ABB RobotStudio station: OpenRobotica_versão16_03_V2.rspag

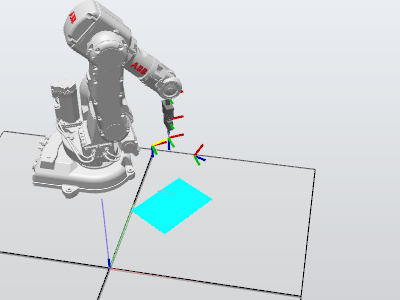
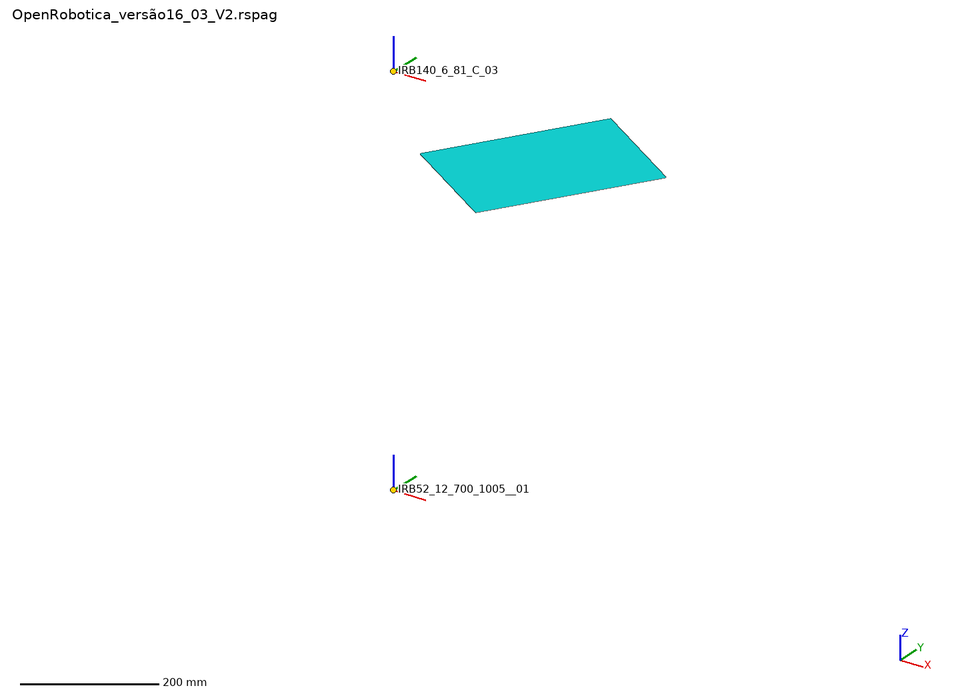
[picture v1: parts stored in the station drawn from their meshes, with robot base, taught points and paths (robot models come from the ABB library and are not in the file)]
--- station ---
Station V1 (saved by RobotStudio 23.2.10395.0)
Controller Robot_ISEP_IRB140, task T_ROB1: task frame (RAPID world) sits at (0, 0, 670) mm in the station
Controller Robot_ISEP_IRB140
  mechanical unit ROB_1: IRB140_6_81_C_03, 6 joints, base frame (0, 0, 0) mm
Controller Robo_open_v2
  mechanical unit ROB_1: IRB52_12_700_1005__01, 6 joints, base frame (0, 0, 0) mm, rotated rx 0 ry 0 rz 90 deg
Layout (positions relative to the parent item):
  - IRB140_6_81_C_03 [mechanism, from %ABB.RobotStudio.Models.IRB140%\IRB140_6_81_C_G_03.rslib] at (0, 0, 670) mm; joint values [0.4681, 0.0159, 0.7824, 0.0025, 0.7739, 3.0595] (rad or m)
  - rob-table [part, from Libraries\rob-table.rslib]
  - pen [mechanism, from Libraries\pen.rslib] at (0, 0, 0) mm
  - paper [part, from Libraries\paper.rslib]
  - IRB52_12_700_1005__01 [mechanism, from %ABB.RobotStudio.Models.IRB52%\IRB52_12_700_1005_G_01.rslib] at (0, 0, 0) mm, rotated rx 0 ry 0 rz 90 deg; joint values [0, 0, 0, 0, 0, 0] (rad or m)
  - A3_Vertical [part] at (450, 125, 790) mm, rotated rx 0 ry 0 rz -90 deg, size 297 x 420 x 0.5 mm
  - A3_Horizontal [part] at (747, 125, 790) mm, rotated rx 0 ry 0 rz 180 deg, size 297 x 420 x 0.5 mm
  - A4_Vertical [part] at (450, 125, 790) mm, rotated rx 0 ry 0 rz -90 deg, size 210 x 297 x 0.5 mm
  - A4_Horizontal [part] at (383.64, -3.77, 703.99) mm, rotated rx -179.83 ry -0.08 rz -32.58 deg, size 210 x 297 x 0.5 mm
  - A5_Vertical [part] at (450, 125, 790) mm, rotated rx 0 ry 0 rz -90 deg, size 148 x 210 x 0.5 mm
  - A5_Horizontal [part] at (450, -85, 790) mm, size 148 x 210 x 0.5 mm
  - MyNewTool [mechanism, from Libraries\Tool_IRB120.rslib] at (304.13, 153.88, 1044.81) mm, rotated rx -179.89 ry 0.07 rz 31.42 deg
Attachment: MyNewTool is attached to IRB140_6_81_C_03 / Link6
Targets, tools, work objects and paths stored in the station and not in the controller backup, written as RAPID:
! task T_ROB1
MODULE Module1
  CONST robtarget Target_Start:=[[0,0,0],[1,0,0,0],[0,0,0,0],[9E+09,9E+09,9E+09,9E+09,9E+09,9E+09]];
ENDMODULE

! task T_ROB1
MODULE DryLetter
  VAR robtarget sup_centro:=[[0,0,0],[1,0,0,0],[0,0,0,0],[9E+09,9E+09,9E+09,9E+09,9E+09,9E+09]];
  VAR robtarget meio_centro:=[[0,0,0],[1,0,0,0],[0,0,0,0],[9E+09,9E+09,9E+09,9E+09,9E+09,9E+09]];
  VAR robtarget inf_centro:=[[0,0,0],[1,0,0,0],[0,0,0,0],[9E+09,9E+09,9E+09,9E+09,9E+09,9E+09]];
  VAR robtarget up_meio_esq:=[[0,0,0],[1,0,0,0],[0,0,0,0],[9E+09,9E+09,9E+09,9E+09,9E+09,9E+09]];
  VAR robtarget sup_dir_meio:=[[0,0,0],[1,0,0,0],[0,0,0,0],[9E+09,9E+09,9E+09,9E+09,9E+09,9E+09]];
  VAR robtarget inf_dir_meio:=[[0,0,0],[1,0,0,0],[0,0,0,0],[9E+09,9E+09,9E+09,9E+09,9E+09,9E+09]];
ENDMODULE

! task T_ROB1
MODULE Math
  PROC impressmenu()
    write_string;
    calculo_size;
    settingsTextMenu;
    settingsPageMenu;
    write_string;
    impress_mecanism;
  ENDPROC
ENDMODULE

! task T_ROB1
MODULE Menu
  PROC start_default()
    WaitTime 3;
  ENDPROC
  PROC principal_menu()
    menu_text;
    menu_paper;
  ENDPROC
  PROC automaticPrinting()
    calculateSizeLetterAutomated;
    calculateOrigin;
    impressMecanism;
  ENDPROC
ENDMODULE

! task T_ROB1
MODULE Fonts
  VAR robtarget target_aMidInf1Esq12:=[[0,0,0],[1,0,0,0],[0,0,0,0],[9E+09,9E+09,9E+09,9E+09,9E+09,9E+09]];
  VAR robtarget target_oMidInf1Esq12:=[[0,0,0],[1,0,0,0],[0,0,0,0],[9E+09,9E+09,9E+09,9E+09,9E+09,9E+09]];
  VAR robtarget target_oMidInf1Dir12:=[[0,0,0],[1,0,0,0],[0,0,0,0],[9E+09,9E+09,9E+09,9E+09,9E+09,9E+09]];
  VAR robtarget target_aMidInf1Dir12:=[[0,0,0],[1,0,0,0],[0,0,0,0],[9E+09,9E+09,9E+09,9E+09,9E+09,9E+09]];
ENDMODULE


--- Backups/Robot_ISEP_IRB140/RAPID/TASK1/PROGMOD/CalibData.mod ---
MODULE CalibData
    PERS tooldata tWeldGun:=[TRUE,[[125.800591275,0,391.268161315],[0.898794046,0,0.438371147,0]],[3,[0,0,100],[0,1,0,0],0,0,0]];
    TASK PERS wobjdata Workobject_Paper:= [FALSE,TRUE,"",[[207.804,202.871,30.7786],[0.000727564,-0.962645,-0.270763,0.000849984]],[[0,0,0],[1,0,0,0]]];

    PERS wobjdata WA5 := [FALSE,TRUE,"",[[207.804,202.871,30.7786],[0.000727564,-0.962645,-0.270763,0.000849984]],[[0,0,0],[1,0,0,0]]];
    PERS wobjdata WA4 := [FALSE,TRUE,"",[[317.336,-107.098,31.058],[0.00324698,-0.996995,0.0772792,0.00429133]],[[0,0,0],[1,0,0,0]]];

    !TASK PERS wobjdata wba4gr3:=[FALSE,TRUE,"",[[317.336,-107.098,31.058],[0.00324698,-0.996995,0.0772792,0.00429133]],[[0,0,0],[1,0,0,0]]];
	!TASK PERS wobjdata wba5gr3:= [FALSE,TRUE,"",[[207.804,202.871,30.7786],[0.000727564,-0.962645,-0.270763,0.000849984]],[[0,0,0],[1,0,0,0]]];


    CONST robtarget Origem:=[[0,0,0],[1,0,0,0],[0,0,0,0],[9E+09,9E+09,9E+09,9E+09,9E+09,9E+09]];
    CONST robtarget Default_position:=[[55,95,-102.5],[1,0,0,0],[0,0,0,0],[9E+09,9E+09,9E+09,9E+09,9E+09,9E+09]];
   ! PERS tooldata pen:=[TRUE,[[0,0,139],[1,0,0,0]],[0.5,[0,0,20],[1,0,0,0],0,0,0]];
    PERS tooldata tcptool:=[TRUE,[[-1.2328,3.617,241.774],[1,0,0,0]],[1,[0,0,125],[1,0,0,0],0,0,0]];
    PERS tooldata pen:=[TRUE,[[0,0,139],[1,0,0,0]],[0.5,[0,0,20],[1,0,0,0],0,0,0]];
    PERS tooldata pen_1:=[TRUE,[[0,0,139],[1,0,0,0]],[0.5,[0,0,20],[1,0,0,0],0,0,0]];
ENDMODULE

--- Backups/Robot_ISEP_IRB140/RAPID/TASK1/PROGMOD/DryLetter.mod ---
MODULE DryLetter
    VAR robtarget up_inf_esq1:=[[0,0,0],[1,0,0,0],[0,0,0,0],[9E+09,9E+09,9E+09,9E+09,9E+09,9E+09]];
    VAR robtarget inf_esq1:=[[0,0,0],[1,0,0,0],[0,0,0,0],[9E+09,9E+09,9E+09,9E+09,9E+09,9E+09]];
    VAR robtarget sup_esq:=[[0,0,0],[1,0,0,0],[0,0,0,0],[9E+09,9E+09,9E+09,9E+09,9E+09,9E+09]];
    VAR robtarget sup_dir:=[[0,0,0],[1,0,0,0],[0,0,0,0],[9E+09,9E+09,9E+09,9E+09,9E+09,9E+09]];
    VAR robtarget inf_dir2:=[[0,0,0],[1,0,0,0],[0,0,0,0],[9E+09,9E+09,9E+09,9E+09,9E+09,9E+09]];
    VAR robtarget up_inf_dir2:=[[0,0,0],[1,0,0,0],[0,0,0,0],[9E+09,9E+09,9E+09,9E+09,9E+09,9E+09]];
    VAR robtarget meio_dir:=[[0,0,0],[1,0,0,0],[0,0,0,0],[9E+09,9E+09,9E+09,9E+09,9E+09,9E+09]];
    VAR robtarget meio_esq:=[[0,0,0],[1,0,0,0],[0,0,0,0],[9E+09,9E+09,9E+09,9E+09,9E+09,9E+09]];
    VAR robtarget up_final:=[[0,0,0],[1,0,0,0],[0,0,0,0],[9E+09,9E+09,9E+09,9E+09,9E+09,9E+09]];
    PROC Path_b()

    ENDPROC
    PROC dry_letter_a()

    ENDPROC
    PROC Letra_A()
        MoveJ up_inf_esq1,v100,fine,tcptool\WObj:=Workobject_Paper;
        MoveL inf_esq1,v100,fine,tcptool\WObj:=Workobject_Paper;
        MoveL sup_esq,v100,z0,tcptool\WObj:=Workobject_Paper;
        MoveL sup_dir,v100,z0,tcptool\WObj:=Workobject_Paper;
        MoveL inf_dir2,v100,fine,tcptool\WObj:=Workobject_Paper;
        MoveL up_inf_dir2,v100,z0,tcptool\WObj:=Workobject_Paper;
        MoveL meio_dir,v100,z0,tcptool\WObj:=Workobject_Paper;
        MoveL meio_esq,v100,fine,tcptool\WObj:=Workobject_Paper;
        MoveL up_final,v100,z0,tcptool\WObj:=Workobject_Paper;
    ENDPROC
    PROC Letra_B()
        MoveJ target_oInf1Esq1,v100,fine,tcptool\WObj:=Workobject_Paper;
        MoveL target_oInf1Esq1,v100,fine,tcptool\WObj:=Workobject_Paper;
        MoveL target_oInf1Esq1,v100,fine,tcptool\WObj:=Workobject_Paper;
    ENDPROC
    PROC Letra_F()
        MoveJ up_inf_esq1,v100,fine,tcptool\WObj:=Workobject_Paper;
    ENDPROC
    PROC Space_letter()
        MoveJ target_oInf1Esq1,v100,fine,tcptool\WObj:=Workobject_Paper;
    ENDPROC
ENDMODULE

--- Backups/Robot_ISEP_IRB140/RAPID/TASK1/PROGMOD/Fonts.mod ---
MODULE Fonts

    ! Offset Z
    VAR num offsetZa := 10;
    VAR num offsetZo := 1;

    ! On the paper

    VAR robtarget target_oInf1Esq1;
    VAR robtarget target_oInf1Esq2;
    VAR robtarget target_oInf1Centro;
    VAR robtarget target_oInf1Dir1;
    VAR robtarget target_oInf1Dir2;

    VAR robtarget target_oInf2Esq1;
    VAR robtarget target_oInf2Esq2;
    VAR robtarget target_oInf2Centro;
    VAR robtarget target_oInf2Dir1;
    VAR robtarget target_oInf2Dir2;

    VAR robtarget target_oCentroEsq1;
    VAR robtarget target_oCentroEsq2;
    VAR robtarget target_oCentroCentro;
    VAR robtarget target_oCentroDir1;
    VAR robtarget target_oCentroDir2;

    VAR robtarget target_oSup1Esq1;
    VAR robtarget target_oSup1Esq2;
    VAR robtarget target_oSup1Centro;
    VAR robtarget target_oSup1Dir1;
    VAR robtarget target_oSup1Dir2;

    VAR robtarget target_oSup2Esq1;
    VAR robtarget target_oSup2Esq2;
    VAR robtarget target_oSup2Centro;
    VAR robtarget target_oSup2Dir1;
    VAR robtarget target_oSup2Dir2;

    ! Above the paper

    VAR robtarget target_aInf1Esq1;
    VAR robtarget target_aInf1Esq2;
    VAR robtarget target_aInf1Centro;
    VAR robtarget target_aInf1Dir1;
    VAR robtarget target_aInf1Dir2;

    VAR robtarget target_aInf2Esq1;
    VAR robtarget target_aInf2Esq2;
    VAR robtarget target_aInf2Centro;
    VAR robtarget target_aInf2Dir1;
    VAR robtarget target_aInf2Dir2;

    VAR robtarget target_aCentroEsq1;
    VAR robtarget target_aCentroEsq2;
    VAR robtarget target_aCentroCentro;
    VAR robtarget target_aCentroDir1;
    VAR robtarget target_aCentroDir2;

    VAR robtarget target_aSup1Esq1;
    VAR robtarget target_aSup1Esq2;
    VAR robtarget target_aSup1Centro;
    VAR robtarget target_aSup1Dir1;
    VAR robtarget target_aSup1Dir2;

    VAR robtarget target_aSup2Esq1;
    VAR robtarget target_aSup2Esq2;
    VAR robtarget target_aSup2Centro;
    VAR robtarget target_aSup2Dir1;
    VAR robtarget target_aSup2Dir2;

    ! Last Position
    VAR robtarget last_position;

    VAR robtarget target_aMidInf1Esq12;
    VAR robtarget target_oMidInf1Esq12 ;
    VAR robtarget target_oMidInf1Dir12;
    VAR robtarget target_aMidInf1Dir12;
    VAR robtarget target_aMidCentro_esq2centro;
    VAR robtarget target_oMidCentro_esq2centro;
    VAR robtarget target_oMidCentro_dirdir1centro;
    VAR robtarget target_aMidCentro_dirdir1centro;

PROC draw( )

       TPWrite "Caracter a Imprimir: " + character;

       target_aInf1Esq1   := Offs(origem, coord_y_letter, coord_x_letter, -offsetZa);
       target_oInf1Esq1   := Offs(origem, coord_y_letter, coord_x_letter, offsetZo);
       target_aInf1Esq2   := Offs(target_aInf1Esq1, 0 , comprimento_letras / 4 , 0);
       target_oInf1Esq2   := Offs(target_oInf1Esq1, 0 , comprimento_letras / 4 , 0);
       target_aInf1Centro := Offs(target_aInf1Esq1, 0 , comprimento_letras / 2 , 0);
       target_oInf1Centro := Offs(target_oInf1Esq1, 0 , comprimento_letras / 2 , 0);
       target_aInf1Dir1   := Offs(target_aInf1Esq1, 0 , comprimento_letras * 3 / 4 , 0);
       target_oInf1Dir1   := Offs(target_oInf1Esq1, 0 , comprimento_letras * 3 / 4 , 0);
       target_aInf1Dir2   := Offs(target_aInf1Esq1, 0 , comprimento_letras , 0);
       target_oInf1Dir2   := Offs(target_oInf1Esq1, 0 , comprimento_letras , 0);


       target_aInf2Esq1   := Offs(target_aInf1Esq1, altura_letras / 4 , 0 , 0);
       target_oInf2Esq1   := Offs(target_oInf1Esq1, altura_letras / 4 , 0 , 0);
       target_aInf2Esq2   := Offs(target_aInf1Esq1, altura_letras / 4 , comprimento_letras / 4 , 0);
       target_oInf2Esq2   := Offs(target_oInf1Esq1, altura_letras / 4 , comprimento_letras / 4 , 0);
       target_aInf2Centro := Offs(target_aInf1Esq1, altura_letras / 4 , comprimento_letras / 2 , 0);
       target_oInf2Centro := Offs(target_oInf1Esq1, altura_letras / 4 , comprimento_letras / 2 , 0);
       target_aInf2Dir1   := Offs(target_aInf1Esq1, altura_letras / 4 , comprimento_letras * 3 / 4 , 0);
       target_oInf2Dir1   := Offs(target_oInf1Esq1, altura_letras / 4 , comprimento_letras * 3 / 4 , 0);
       target_aInf2Dir2   := Offs(target_aInf1Esq1, altura_letras / 4 , comprimento_letras , 0);
       target_oInf2Dir2   := Offs(target_oInf1Esq1, altura_letras / 4 , comprimento_letras , 0);


       target_aCentroEsq1   := Offs(target_aInf1Esq1, altura_letras / 2 , 0 , 0);
       target_oCentroEsq1   := Offs(target_oInf1Esq1, altura_letras / 2 , 0 , 0);
       target_aCentroEsq2   := Offs(target_aInf1Esq1, altura_letras / 2 , comprimento_letras / 4 , 0);
       target_oCentroEsq2   := Offs(target_oInf1Esq1, altura_letras / 2 , comprimento_letras / 4 , 0);
       target_aCentroCentro := Offs(target_aInf1Esq1, altura_letras / 2 , comprimento_letras / 2 , 0);
       target_oCentroCentro := Offs(target_oInf1Esq1, altura_letras / 2 , comprimento_letras / 2 , 0);
       target_aCentroDir1   := Offs(target_aInf1Esq1, altura_letras / 2 , comprimento_letras * 3 / 4 , 0);
       target_oCentroDir1   := Offs(target_oInf1Esq1, altura_letras / 2 , comprimento_letras * 3 / 4 , 0);
       target_aCentroDir2   := Offs(target_aInf1Esq1, altura_letras / 2 , comprimento_letras , 0);
       target_oCentroDir2   := Offs(target_oInf1Esq1, altura_letras / 2 , comprimento_letras , 0);

       target_aSup2Esq1   := Offs(target_aInf1Esq1, altura_letras * 3 / 4 , 0 , 0);
       target_oSup2Esq1   := Offs(target_oInf1Esq1, altura_letras * 3 / 4 , 0 , 0);
       target_aSup2Esq2   := Offs(target_aInf1Esq1, altura_letras * 3 / 4 , comprimento_letras / 4 , 0);
       target_oSup2Esq2   := Offs(target_oInf1Esq1, altura_letras * 3 / 4 , comprimento_letras / 4 , 0);
       target_aSup2Centro := Offs(target_aInf1Esq1, altura_letras * 3 / 4 , comprimento_letras / 2 , 0);
       target_oSup2Centro := Offs(target_oInf1Esq1, altura_letras * 3 / 4 , comprimento_letras / 2 , 0);
       target_aSup2Dir1   := Offs(target_aInf1Esq1, altura_letras * 3 / 4 , comprimento_letras * 3 / 4 , 0);
       target_oSup2Dir1   := Offs(target_oInf1Esq1, altura_letras * 3 / 4 , comprimento_letras * 3 / 4 , 0);
       target_aSup2Dir2   := Offs(target_aInf1Esq1, altura_letras * 3 / 4 , comprimento_letras , 0);
       target_oSup2Dir2   := Offs(target_oInf1Esq1, altura_letras * 3 / 4 , comprimento_letras , 0);

       target_aSup1Esq1   := Offs(target_aInf1Esq1, altura_letras , 0 , 0);
       target_oSup1Esq1   := Offs(target_oInf1Esq1, altura_letras , 0 , 0);
       target_aSup1Esq2   := Offs(target_aInf1Esq1, altura_letras , comprimento_letras / 4 , 0);
       target_oSup1Esq2   := Offs(target_oInf1Esq1, altura_letras , comprimento_letras / 4 , 0);
       target_aSup1Centro := Offs(target_aInf1Esq1, altura_letras , comprimento_letras / 2 , 0);
       target_oSup1Centro := Offs(target_oInf1Esq1, altura_letras , comprimento_letras / 2 , 0);
       target_aSup1Dir1   := Offs(target_aInf1Esq1, altura_letras , comprimento_letras * 3 / 4 , 0);
       target_oSup1Dir1   := Offs(target_oInf1Esq1, altura_letras , comprimento_letras * 3 / 4 , 0);
       target_aSup1Dir2   := Offs(target_aInf1Esq1, altura_letras , comprimento_letras , 0);
       target_oSup1Dir2   := Offs(target_oInf1Esq1, altura_letras , comprimento_letras , 0);

       IF "Classic" = text_FontType THEN
	        IF "A" = character OR "a" = character THEN

                    ! adaptar origem

                    MoveJ target_aInf1Esq1, v100, fine, tcptool\WObj:=Workobject_Paper;
                    MoveL target_oInf1Esq1, v100, fine, tcptool\WObj:=Workobject_Paper;
                    MoveL target_oSup1Esq1, v100, z50, tcptool\WObj:=Workobject_Paper;
                    MoveL target_oSup1Dir2, v100, z50, tcptool\WObj:=Workobject_Paper;
                    MoveL target_oInf1Dir2, v100, fine, tcptool\WObj:=Workobject_Paper;
                    MoveL target_oCentroDir2, v100, z0, tcptool\WObj:=Workobject_Paper;
                    MoveL target_oCentroEsq1, v100, fine, tcptool\WObj:=Workobject_Paper;
                    MoveL target_aCentroEsq1, v100, fine, tcptool\WObj:=Workobject_Paper;

                    !last_position := CRobT(\Tool:=tcptool\WObj:=Workobject_Paper);

	        ELSEIF "B" = character OR "b" = character THEN

                ! definição Trajeto

                MoveJ target_oInf1Esq1, v100, fine, tcptool\WObj:=Workobject_Paper;
                MoveL target_oInf1Esq1, v100, fine, tcptool\WObj:=Workobject_Paper;
                MoveL target_oSup1Esq1, v100, fine, tcptool\WObj:=Workobject_Paper;
                MoveL target_oSup1Centro, v100, z0, tcptool\WObj:=Workobject_Paper;
                MoveC target_oSup2Dir2, target_oCentroCentro, v100, fine, tcptool\WObj:=Workobject_Paper;
                MoveL target_oCentroEsq1, v100, fine, tcptool\WObj:=Workobject_Paper;
                MoveL target_oCentroCentro, v100, fine, tcptool\WObj:=Workobject_Paper;
                MoveC target_oInf2Dir2 ,target_oInf1Centro, v100, fine, tcptool\WObj:=Workobject_Paper;
                MoveL target_oInf1Esq1, v100, fine, tcptool\WObj:=Workobject_Paper;

                MoveL target_aInf1Esq1, v100, z0, tcptool\WObj:=Workobject_Paper;

                last_position := CRobT(\Tool:=tcptool\WObj:=Workobject_Paper);

	        ELSEIF "C" = character OR "c" = character THEN

                MoveJ target_aInf2Dir2, v100, fine, tcptool\WObj:=Workobject_Paper;
                MoveL target_oInf2Dir2, v100, fine, tcptool\WObj:=Workobject_Paper;
                MoveC target_oInf1Centro, target_oInf2Esq1, v100, fine, tcptool\WObj:=Workobject_Paper;
                MoveL target_oSup2Esq1, v100, fine, tcptool\WObj:=Workobject_Paper;
                MoveC target_oSup1Centro, target_oSup2Dir2, v100, fine, tcptool\WObj:=Workobject_Paper;
                MoveL target_aSup1Centro, v100, fine, tcptool\WObj:=Workobject_Paper;


	        ELSEIF "D" = character OR "d" = character THEN
	            ! Instructions to draw letter "D"
                MoveJ target_aInf1Esq1, v100, fine, tcptool\WObj:=Workobject_Paper;
                MoveL target_oInf1Esq1, v100, fine, tcptool\WObj:=Workobject_Paper;
                MoveL target_oSup1Esq1, v100, fine, tcptool\WObj:=Workobject_Paper;
                MoveL target_oSup1Dir2, v100, z200, tcptool\WObj:=Workobject_Paper;
                MoveL target_oInf1Dir2, v100, z200, tcptool\WObj:=Workobject_Paper;
                MoveL target_oInf1Esq1, v100, fine, tcptool\WObj:=Workobject_Paper;
                MoveL target_aInf1Esq1, v100, fine, tcptool\WObj:=Workobject_Paper;

	        ELSEIF "E" = character OR "e" = character THEN
	            ! Instructions to draw letter "E"
                MoveJ target_aInf1Dir2, v100, fine, tcptool\WObj:=Workobject_Paper;
                MoveL target_oInf1Dir2, v100, fine, tcptool\WObj:=Workobject_Paper;
                MoveL target_oInf1Esq1, v100, fine, tcptool\WObj:=Workobject_Paper;
                MoveL target_oSup1Esq1, v100, fine, tcptool\WObj:=Workobject_Paper;
                MoveL target_oSup1Dir2, v100, fine, tcptool\WObj:=Workobject_Paper;
                MoveL target_aSup1Dir2, v100, fine, tcptool\WObj:=Workobject_Paper;
                MoveL target_aCentroEsq1, v100, fine, tcptool\WObj:=Workobject_Paper;
                MoveL target_oCentroEsq1, v100, fine, tcptool\WObj:=Workobject_Paper;
                MoveL target_oCentroCentro, v100, fine, tcptool\WObj:=Workobject_Paper;
                MoveL target_aCentroCentro, v100, fine, tcptool\WObj:=Workobject_Paper;

	        ELSEIF "F" = character OR "f" = character THEN
	            ! Instructions to draw letter "F"
                MoveJ target_aInf1Esq1, v100, fine, tcptool\WObj:=Workobject_Paper;
                MoveL target_oInf1Esq1, v100, fine, tcptool\WObj:=Workobject_Paper;
                MoveL target_oSup1Esq1, v100, fine, tcptool\WObj:=Workobject_Paper;
                MoveL target_oSup1Dir2, v100, fine, tcptool\WObj:=Workobject_Paper;
                MoveL target_aSup1Dir2, v100, fine, tcptool\WObj:=Workobject_Paper;
                MoveL target_aCentroEsq1, v100, fine, tcptool\WObj:=Workobject_Paper;
                MoveL target_oCentroEsq1, v100, fine, tcptool\WObj:=Workobject_Paper;
                MoveL target_oCentroCentro, v100, fine, tcptool\WObj:=Workobject_Paper;
                MoveL target_aCentroCentro, v100, fine, tcptool\WObj:=Workobject_Paper;

	        ELSEIF "G" = character OR "g" = character THEN
	            ! Instructions to draw letter "G"
                !MoveJ target_aInf1Esq1, v100, fine, tcptool\WObj:=Workobject_Paper;
                MoveJ target_aCentroCentro, v100, fine, tcptool\WObj:=Workobject_Paper;
                MoveL target_oCentroCentro, v100, fine, tcptool\WObj:=Workobject_Paper;
                MoveL target_oCentroDir2, v100, fine, tcptool\WObj:=Workobject_Paper;
                MoveL target_oInf1Dir2, v100, fine, tcptool\WObj:=Workobject_Paper;
                MoveL target_oInf1Esq1, v100, z200, tcptool\WObj:=Workobject_Paper;
                MoveL target_oSup2Esq1, v100, fine, tcptool\WObj:=Workobject_Paper;
                MoveC target_oSup1Centro, target_oSup2Dir2, v100, fine, tcptool\WObj:=Workobject_Paper;
                MoveL target_aSup2Dir2, v100, fine, tcptool\WObj:=Workobject_Paper;

	        ELSEIF "H" = character OR "h" = character THEN
	            ! Instructions to draw letter "H"
                MoveJ target_aInf1Esq1, v100, fine, tcptool\WObj:=Workobject_Paper;
                MoveL target_oInf1Esq1, v100, fine, tcptool\WObj:=Workobject_Paper;
                MoveL target_oSup1Esq1, v100, fine, tcptool\WObj:=Workobject_Paper;
                MoveL target_aSup1Esq1, v100, fine, tcptool\WObj:=Workobject_Paper;
                MoveL target_aSup1Dir2, v100, fine, tcptool\WObj:=Workobject_Paper;
                MoveL target_oSup1Dir2, v100, fine, tcptool\WObj:=Workobject_Paper;
                MoveL target_oInf1Dir2, v100, fine, tcptool\WObj:=Workobject_Paper;
                MoveL target_aInf1Dir2, v100, fine, tcptool\WObj:=Workobject_Paper;
                MoveL target_aCentroEsq1, v100, fine, tcptool\WObj:=Workobject_Paper;
                MoveL target_oCentroEsq1, v100, fine, tcptool\WObj:=Workobject_Paper;
                MoveL target_oCentroDir2, v100, fine, tcptool\WObj:=Workobject_Paper;
                MoveL target_aCentroDir2, v100, fine, tcptool\WObj:=Workobject_Paper;

	        ELSEIF "I" = character OR "i" = character THEN
	            ! Instructions to draw letter "I"
                !MoveJ target_aSup1Esq1, v100, fine, tcptool\WObj:=Workobject_Paper;
                MoveJ target_aSup1Centro, v100, fine, tcptool\WObj:=Workobject_Paper;
                MoveL target_oSup1Centro, v100, fine, tcptool\WObj:=Workobject_Paper;
                MoveL target_oInf1Centro, v100, fine, tcptool\WObj:=Workobject_Paper;
                MoveL target_aInf1Centro, v100, fine, tcptool\WObj:=Workobject_Paper;

	        ELSEIF "J" = character OR "j" = character THEN
	            ! Instructions to draw letter "J"
                MoveJ target_aSup1Dir2, v100, fine, tcptool\WObj:=Workobject_Paper;
                MoveL target_oSup1Dir2, v100, fine, tcptool\WObj:=Workobject_Paper;
                MoveL target_oInf2Dir2, v100, fine, tcptool\WObj:=Workobject_Paper;
                MoveC target_oInf1Centro, target_oInf2Esq1, v100, fine, tcptool\WObj:=Workobject_Paper;
                MoveL target_aInf2Esq1, v100, fine, tcptool\WObj:=Workobject_Paper;

	        ELSEIF "K" = character OR "k" = character THEN
	            ! Instructions to draw letter "K"
                MoveJ target_aInf1Esq1, v100, fine, tcptool\WObj:=Workobject_Paper;
                MoveL target_oInf1Esq1, v100, fine, tcptool\WObj:=Workobject_Paper;
                MoveL target_oSup1Esq1, v100, fine, tcptool\WObj:=Workobject_Paper;
                MoveL target_aSup1Esq1, v100, fine, tcptool\WObj:=Workobject_Paper;
                MoveL target_aCentroEsq1, v100, fine, tcptool\WObj:=Workobject_Paper;
                MoveL target_oCentroEsq1, v100, fine, tcptool\WObj:=Workobject_Paper;
                MoveL target_oSup1Dir2, v100, fine, tcptool\WObj:=Workobject_Paper;
                MoveL target_aSup1Dir2, v100, fine, tcptool\WObj:=Workobject_Paper;
                MoveL target_aCentroEsq1, v100, fine, tcptool\WObj:=Workobject_Paper;
                MoveL target_oCentroEsq1, v100, fine, tcptool\WObj:=Workobject_Paper;
                MoveL target_oInf1Dir2, v100, fine, tcptool\WObj:=Workobject_Paper;
                MoveL target_aInf1Dir2, v100, fine, tcptool\WObj:=Workobject_Paper;

	        ELSEIF "L" = character OR "l" = character THEN
	            ! Instructions to draw letter "L"
                MoveJ target_aSup1Esq1, v100, fine, tcptool\WObj:=Workobject_Paper;
                MoveL target_oSup1Esq1, v100, fine, tcptool\WObj:=Workobject_Paper;
                MoveL target_oInf1Esq1, v100, fine, tcptool\WObj:=Workobject_Paper;
                MoveL target_oInf1Dir2, v100, fine, tcptool\WObj:=Workobject_Paper;
                MoveL target_aInf1Dir2, v100, fine, tcptool\WObj:=Workobject_Paper;

	       ELSEIF "M" = character OR "m" = character THEN
	            ! Instructions to draw letter "M"

		        ! Movement
		        MoveJ target_aInf1Esq1, v100, fine, tcptool\WObj:=Workobject_Paper;
		        MoveL target_oInf1Esq1, v100, fine, tcptool\WObj:=Workobject_Paper;
		        MoveL target_oSup1Esq1, v100, fine, tcptool\WObj:=Workobject_Paper;
		        MoveL target_oCentroCentro, v100, fine, tcptool\WObj:=Workobject_Paper;
		        MoveL target_oSup1Dir2, v100, fine, tcptool\WObj:=Workobject_Paper;
		        MoveL target_oInf1Dir2, v100, fine, tcptool\WObj:=Workobject_Paper;
		        MoveL target_aInf1Dir2, v100, fine, tcptool\WObj:=Workobject_Paper;

	        ELSEIF "N" = character OR "n" = character THEN
		        ! Movement
		        MoveJ target_aInf1Esq1, v100, fine, tcptool\WObj:=Workobject_Paper;
		        MoveL target_oInf1Esq1, v100, fine, tcptool\WObj:=Workobject_Paper;
		        MoveL target_oSup1Esq1, v100, fine, tcptool\WObj:=Workobject_Paper;
		        MoveL target_oInf1Dir2, v100, fine, tcptool\WObj:=Workobject_Paper;
		        MoveL target_oSup1Dir2, v100, fine, tcptool\WObj:=Workobject_Paper;
		        MoveL target_aSup1Dir2, v100, fine, tcptool\WObj:=Workobject_Paper;

	        ELSEIF "O" = character OR "o" = character THEN

		        MoveJ target_aInf2Esq1, v100, fine, tcptool\WObj:=Workobject_Paper;
                MoveL target_oInf2Esq1, v100, fine, tcptool\WObj:=Workobject_Paper;
                MoveL target_oSup2Esq1, v100, fine, tcptool\WObj:=Workobject_Paper;
                MoveC target_oSup1Centro, target_oSup2Dir2, v100, fine, tcptool\WObj:=Workobject_Paper;
                MoveL target_oInf2Dir2, v100, fine, tcptool\WObj:=Workobject_Paper;
                MoveC target_oInf1Centro, target_oInf2Esq1, v100, fine, tcptool\WObj:=Workobject_Paper;
                MoveL target_aInf2Esq1, v100, fine, tcptool\WObj:=Workobject_Paper;

	        ELSEIF "P" = character OR "p" = character THEN

		        ! Movement
		        MoveJ target_aInf1Esq1, v100, fine, tcptool\WObj:=Workobject_Paper;
		        MoveL target_oInf1Esq1, v100, fine, tcptool\WObj:=Workobject_Paper;
		        MoveL target_oSup1Esq1, v100, fine, tcptool\WObj:=Workobject_Paper;
		        MoveL target_oSup1Centro, v100, fine, tcptool\WObj:=Workobject_Paper;
		        MoveC target_oSup2Dir2 , target_oCentroEsq2 , v100, fine, tcptool\WObj:=Workobject_Paper;
		        MoveL target_oCentroCentro, v100, fine, tcptool\WObj:=Workobject_Paper;
		        MoveL target_aCentroEsq1, v100, fine, tcptool\WObj:=Workobject_Paper;


	        ELSEIF "Q" = character OR "q" = character THEN
	            ! Instructions to draw letter "Q"
                MoveJ target_aInf2Esq1, v100, fine, tcptool\WObj:=Workobject_Paper;
                MoveL target_oInf2Esq1, v100, fine, tcptool\WObj:=Workobject_Paper;
                MoveL target_oSup2Esq1, v100, fine, tcptool\WObj:=Workobject_Paper;
                MoveC target_oSup1Centro, target_oSup2Dir2, v100, fine, tcptool\WObj:=Workobject_Paper;
                MoveL target_oInf2Dir2, v100, fine, tcptool\WObj:=Workobject_Paper;
                MoveC target_oInf1Centro, target_oInf2Esq1, v100, fine, tcptool\WObj:=Workobject_Paper;
                MoveL target_aInf2Esq1, v100, fine, tcptool\WObj:=Workobject_Paper;
                MoveL target_aInf2Dir1, v100, fine, tcptool\WObj:=Workobject_Paper;
                MoveL target_oInf2Dir1, v100, fine, tcptool\WObj:=Workobject_Paper;
                MoveL target_oInf1Dir2, v100, fine, tcptool\WObj:=Workobject_Paper;
                MoveL target_aInf1Dir2, v100, fine, tcptool\WObj:=Workobject_Paper;

	        ELSEIF "R" = character OR "r" = character THEN
	            ! Instructions to draw letter "R"
                MoveJ target_aInf1Esq1, v100, fine, tcptool\WObj:=Workobject_Paper;
                MoveL target_oInf1Esq1, v100, fine, tcptool\WObj:=Workobject_Paper;
                MoveL target_oSup1Esq1, v100, fine, tcptool\WObj:=Workobject_Paper;
                MoveL target_oSup1Centro, v100, fine, tcptool\WObj:=Workobject_Paper;
                MoveC target_oSup2Dir2 , target_oCentroCentro , v100, fine, tcptool\WObj:=Workobject_Paper;
                MoveL target_oCentroEsq1, v100, fine, tcptool\WObj:=Workobject_Paper;
                MoveL target_oInf1Dir2, v100, fine, tcptool\WObj:=Workobject_Paper;
                MoveL target_aInf1Dir2, v100, fine, tcptool\WObj:=Workobject_Paper;

	        ELSEIF "S" = character OR "s" = character THEN
	            ! Instructions to draw letter "S"

		        ! Movement
		        MoveJ target_aSup2Dir2, v100, fine, tcptool\WObj:=Workobject_Paper;
		        MoveL target_oSup2Dir2, v100, fine, tcptool\WObj:=Workobject_Paper;
		        MoveC target_oSup1Centro , target_oSup2Esq1 , v100, fine, tcptool\WObj:=Workobject_Paper;

                MoveL target_oCentroEsq1, v100, z150, tcptool\WObj:=Workobject_Paper;
                MoveL target_oCentroCentro, v100, fine, tcptool\WObj:=Workobject_Paper;
                MoveL target_oCentroDir2, v100, z150, tcptool\WObj:=Workobject_Paper;
                MoveL target_oInf2Dir2, v100, fine, tcptool\WObj:=Workobject_Paper;

                MoveC target_oInf1Centro , target_oInf2Esq1 , v100, fine, tcptool\WObj:=Workobject_Paper;
		        MoveL target_aInf2Esq1, v100, fine, tcptool\WObj:=Workobject_Paper;


	        ELSEIF "T" = character OR "t" = character THEN
	            ! Instructions to draw letter "T"
                target_aInf1Centro := Offs( target_aInf1Esq1 , 0 , comprimento_letras/2 , 0);
                target_oInf1Centro := Offs( target_oInf1Esq1 , 0 , comprimento_letras/2 , 0);
                target_aSup1Centro := Offs( target_aInf1Esq1 , altura_letras , comprimento_letras/2 , 0);
                target_oSup1Centro := Offs( target_oInf1Esq1 , altura_letras , comprimento_letras/2 , 0);

		        ! Movement
		        MoveJ target_aSup1Esq1, v100, fine, tcptool\WObj:=Workobject_Paper;
		        MoveL target_oSup1Esq1, v100, fine, tcptool\WObj:=Workobject_Paper;
		        MoveL target_oSup1Dir2, v100, fine, tcptool\WObj:=Workobject_Paper;
		        MoveL target_oSup1Centro, v100, fine, tcptool\WObj:=Workobject_Paper;
		        MoveL target_oInf1Centro, v100, fine, tcptool\WObj:=Workobject_Paper;
		        MoveL target_aInf1Centro, v100, fine, tcptool\WObj:=Workobject_Paper;

	        ELSEIF "U" = character OR "u" = character THEN

		        ! Movement
		        MoveJ target_aSup1Esq1, v100, fine, tcptool\WObj:=Workobject_Paper;
		        MoveL target_oSup1Esq1, v100, fine, tcptool\WObj:=Workobject_Paper;
		        MoveL target_oInf2Esq1, v100, fine, tcptool\WObj:=Workobject_Paper;
		        MoveC target_oInf1Centro , target_oInf2Dir2 , v100, fine, tcptool\WObj:=Workobject_Paper;
		        MoveL target_oSup1Dir2, v100, fine, tcptool\WObj:=Workobject_Paper;
		        MoveL target_aSup1Dir2, v100, fine, tcptool\WObj:=Workobject_Paper;


	        ELSEIF "V" = character OR "v" = character THEN

		        ! Movement
		        MoveJ target_aSup1Esq1, v100, fine, tcptool\WObj:=Workobject_Paper;
		        MoveL target_oSup1Esq1, v100, fine, tcptool\WObj:=Workobject_Paper;
		        MoveL target_oInf1Centro, v100, fine, tcptool\WObj:=Workobject_Paper;
		        MoveL target_oSup1Dir2, v100, fine, tcptool\WObj:=Workobject_Paper;
		        MoveL target_aSup1Dir2, v100, fine, tcptool\WObj:=Workobject_Paper;
		        !MoveL target_aInf1Dir2, v100, fine, tcptool\WObj:=Workobject_Paper;

	        ELSEIF "W" = character OR "w" = character THEN


		        ! Movement
		        MoveJ target_aSup1Esq1, v100, fine, tcptool\WObj:=Workobject_Paper;
		        MoveL target_oSup1Esq1, v100, fine, tcptool\WObj:=Workobject_Paper;
		        MoveL target_oInf1Esq2, v100, fine, tcptool\WObj:=Workobject_Paper;
		        MoveL target_oCentroCentro, v100, fine, tcptool\WObj:=Workobject_Paper;
		        MoveL target_oInf1Dir1, v100, fine, tcptool\WObj:=Workobject_Paper;
		        MoveL target_oSup1Dir2, v100, fine, tcptool\WObj:=Workobject_Paper;
		        MoveL target_aSup1Dir2, v100, fine, tcptool\WObj:=Workobject_Paper;
		        !MoveL target_aInf1Dir2, v100, fine, tcptool\WObj:=Workobject_Paper;

	        ELSEIF "X" = character OR "x" = character THEN
	            ! Instructions to draw letter "X"

		        ! Movement
		        MoveJ target_aSup1Esq1, v100, fine, tcptool\WObj:=Workobject_Paper;
		        MoveL target_oSup1Esq1, v100, fine, tcptool\WObj:=Workobject_Paper;
		        MoveL target_oInf1Dir2, v100, fine, tcptool\WObj:=Workobject_Paper;
		        MoveL target_aInf1Dir2, v100, fine, tcptool\WObj:=Workobject_Paper;
		        MoveL target_aSup1Dir2, v100, fine, tcptool\WObj:=Workobject_Paper;
		        MoveL target_oSup1Dir2, v100, fine, tcptool\WObj:=Workobject_Paper;
		        MoveL target_oInf1Esq1, v100, fine, tcptool\WObj:=Workobject_Paper;
		        MoveL target_aInf1Esq1, v100, fine, tcptool\WObj:=Workobject_Paper;
		        !MoveL target_aInf1Dir2, v100, fine, tcptool\WObj:=Workobject_Paper;

	        ELSEIF "Y" = character OR "y" = character THEN

		        ! Movement
		        MoveJ target_aSup1Esq1, v100, fine, tcptool\WObj:=Workobject_Paper;
		        MoveL target_oSup1Esq1, v100, fine, tcptool\WObj:=Workobject_Paper;
		        MoveL target_oCentroCentro, v100, fine, tcptool\WObj:=Workobject_Paper;
		        MoveL target_oSup1Dir2, v100, fine, tcptool\WObj:=Workobject_Paper;
		        MoveL target_aSup1Dir2, v100, fine, tcptool\WObj:=Workobject_Paper;
		        MoveL target_aCentroCentro, v100, fine, tcptool\WObj:=Workobject_Paper;
		        MoveL target_oCentroCentro, v100, fine, tcptool\WObj:=Workobject_Paper;
		        MoveL target_oInf1Centro, v100, fine, tcptool\WObj:=Workobject_Paper;
		        MoveL target_aInf1Centro, v100, fine, tcptool\WObj:=Workobject_Paper;
		        !MoveL target_aInf1Dir2, v100, fine, tcptool\WObj:=Workobject_Paper;

	        ELSEIF "Z" = character OR "z" = character THEN
	           ! Instructions to draw letter "Z"

		        ! Movement
		        MoveJ target_aSup1Esq1, v100, fine, tcptool\WObj:=Workobject_Paper;
		        MoveL target_oSup1Esq1, v100, fine, tcptool\WObj:=Workobject_Paper;
		        MoveL target_oSup1Dir2, v100, fine, tcptool\WObj:=Workobject_Paper;
		        MoveL target_oInf1Esq1, v100, fine, tcptool\WObj:=Workobject_Paper;
		        MoveL target_oInf1Dir2, v100, fine, tcptool\WObj:=Workobject_Paper;
		        MoveL target_aInf1Dir2, v100, fine, tcptool\WObj:=Workobject_Paper;

	        ELSEIF " " = character THEN
	            ! Instructions to draw letter " "
                MoveJ target_aInf1Esq1, v100, fine, tcptool\WObj:=Workobject_Paper;

            ELSEIF "0" = character THEN
                MoveJ target_aInf2Esq1, v100, fine, tcptool\WObj:=Workobject_Paper;
                MoveL target_oInf2Esq1, v100, fine, tcptool\WObj:=Workobject_Paper;
                MoveL target_oSup2Esq1, v100, fine, tcptool\WObj:=Workobject_Paper;
                MoveC target_oSup1Centro, target_oSup2Dir2, v100, fine, tcptool\WObj:=Workobject_Paper;
                MoveL target_oInf2Dir2, v100, fine, tcptool\WObj:=Workobject_Paper;
                MoveC target_oInf1Centro, target_oInf2Esq1, v100, fine, tcptool\WObj:=Workobject_Paper;
                MoveL target_aInf2Esq1, v100, fine, tcptool\WObj:=Workobject_Paper;
                MoveL target_aInf2Esq2, v100, fine, tcptool\WObj:=Workobject_Paper;
                MoveL target_oInf2Esq2, v100, fine, tcptool\WObj:=Workobject_Paper;
                MoveL target_oSup2Dir1, v100, fine, tcptool\WObj:=Workobject_Paper;
                MoveL target_aSup2Dir1, v100, fine, tcptool\WObj:=Workobject_Paper;

            ELSEIF "1" = character THEN
                MoveJ target_aSup2Esq2, v100, fine, tcptool\WObj:=Workobject_Paper;
                MoveL target_oSup2Esq2, v100, fine, tcptool\WObj:=Workobject_Paper;
                MoveL target_oSup1Centro, v100, fine, tcptool\WObj:=Workobject_Paper;
                MoveL target_oInf1Centro, v100, fine, tcptool\WObj:=Workobject_Paper;
                MoveL target_aInf1Centro, v100, fine, tcptool\WObj:=Workobject_Paper;
                MoveL target_aInf1Esq1, v100, fine, tcptool\WObj:=Workobject_Paper;
                MoveL target_oInf1Esq1, v100, fine, tcptool\WObj:=Workobject_Paper;
                MoveL target_oInf1Dir2, v100, fine, tcptool\WObj:=Workobject_Paper;


            ELSEIF "2" = character THEN
                MoveJ target_aSup2Esq1, v100, fine, tcptool\WObj:=Workobject_Paper;
                MoveL target_oSup2Esq1, v100, fine, tcptool\WObj:=Workobject_Paper;
                MoveC target_oSup1Centro, target_oSup2Dir2, v100, fine, tcptool\WObj:=Workobject_Paper;
                MoveL target_oInf1Esq1, v100, fine, tcptool\WObj:=Workobject_Paper;
                MoveL target_oInf1Dir2, v100, fine, tcptool\WObj:=Workobject_Paper;
                MoveL target_aInf1Dir2, v100, fine, tcptool\WObj:=Workobject_Paper;

            ELSEIF "3" = character THEN
                MoveJ target_aSup1Esq2, v100, fine, tcptool\WObj:=Workobject_Paper;
                MoveL target_oSup1Esq2, v100, fine, tcptool\WObj:=Workobject_Paper;
                MoveL target_oSup1Centro, v100, fine, tcptool\WObj:=Workobject_Paper;
                MoveC target_oSup2Dir2, target_oCentroCentro, v100, fine, tcptool\WObj:=Workobject_Paper;
                MoveC target_oInf2Dir2, target_oInf1Centro, v100, fine, tcptool\WObj:=Workobject_Paper;
                MoveL target_oInf1Esq2, v100, fine, tcptool\WObj:=Workobject_Paper;
                MoveL target_aInf1Esq2, v100, fine, tcptool\WObj:=Workobject_Paper;

            ELSEIF "4" = character THEN
                MoveJ target_aInf1Dir1, v100, fine, tcptool\WObj:=Workobject_Paper;
                MoveL target_oInf1Dir1, v100, fine, tcptool\WObj:=Workobject_Paper;
                MoveL target_oSup1Dir1, v100, fine, tcptool\WObj:=Workobject_Paper;
                MoveL target_oSup1Dir1, v100, fine, tcptool\WObj:=Workobject_Paper;
                MoveL target_oInf2Esq1, v100, fine, tcptool\WObj:=Workobject_Paper;
                MoveL target_oInf2Dir2, v100, fine, tcptool\WObj:=Workobject_Paper;
                MoveL target_aInf2Dir2, v100, fine, tcptool\WObj:=Workobject_Paper;


            ELSEIF "5" = character THEN
                MoveJ target_aSup1Dir2, v100, fine, tcptool\WObj:=Workobject_Paper;
                MoveL target_oSup1Dir2, v100, fine, tcptool\WObj:=Workobject_Paper;
                MoveL target_oSup1Esq1, v100, fine, tcptool\WObj:=Workobject_Paper;
                MoveL target_oCentroEsq1, v100, fine, tcptool\WObj:=Workobject_Paper;
                MoveL target_oCentroCentro, v100, fine, tcptool\WObj:=Workobject_Paper;
                MoveC target_oInf2Dir2, target_oInf1Centro, v100, fine, tcptool\WObj:=Workobject_Paper;
                MoveL target_oInf1Esq1, v100, fine, tcptool\WObj:=Workobject_Paper;
                MoveL target_aInf1Esq1, v100, fine, tcptool\WObj:=Workobject_Paper;


            ELSEIF "6" = character THEN
                MoveJ target_aInf2Esq1, v100, fine, tcptool\WObj:=Workobject_Paper;
                MoveL target_oInf2Esq1, v100, fine, tcptool\WObj:=Workobject_Paper;
                MoveC target_oCentroCentro, target_oInf2Dir2, v100, fine, tcptool\WObj:=Workobject_Paper;
                MoveC target_oInf1Centro, target_oInf2Esq1, v100, fine, tcptool\WObj:=Workobject_Paper;
                MoveL target_oSup1Centro, v100, fine, tcptool\WObj:=Workobject_Paper;
                MoveL target_aSup1Centro, v100, fine, tcptool\WObj:=Workobject_Paper;

            ELSEIF "7" = character THEN
                MoveJ target_aInf1Esq1, v100, fine, tcptool\WObj:=Workobject_Paper;
                MoveL target_oInf1Esq1, v100, fine, tcptool\WObj:=Workobject_Paper;
                MoveL target_oSup1Dir2, v100, fine, tcptool\WObj:=Workobject_Paper;
                MoveL target_oSup1Esq1, v100, fine, tcptool\WObj:=Workobject_Paper;
                MoveL target_aSup1Esq1, v100, fine, tcptool\WObj:=Workobject_Paper;

            ELSEIF "8" = character THEN
                MoveJ target_aCentroCentro, v100, fine, tcptool\WObj:=Workobject_Paper;
                MoveL target_oCentroCentro, v100, fine, tcptool\WObj:=Workobject_Paper;
                MoveC target_oInf2Dir2, target_oInf1Centro , v100, fine, tcptool\WObj:=Workobject_Paper;
                MoveC target_oInf2Esq1, target_oCentroCentro , v100, fine, tcptool\WObj:=Workobject_Paper;
                MoveC target_oSup2Esq1, target_oSup1Centro , v100, fine, tcptool\WObj:=Workobject_Paper;
                MoveC target_oSup2Dir2, target_oCentroCentro , v100, fine, tcptool\WObj:=Workobject_Paper;
                MoveL target_aCentroCentro, v100, fine, tcptool\WObj:=Workobject_Paper;

            ELSEIF "9" = character THEN
                MoveJ target_aSup2Dir2, v100, fine, tcptool\WObj:=Workobject_Paper;
                MoveL target_oSup2Dir2, v100, fine, tcptool\WObj:=Workobject_Paper;
                MoveC target_oCentroCentro, target_oSup2Esq1 , v100, fine, tcptool\WObj:=Workobject_Paper;
                MoveC target_oSup1Centro, target_oSup2Dir2 , v100, fine, tcptool\WObj:=Workobject_Paper;
                MoveL target_oInf1Centro, v100, fine, tcptool\WObj:=Workobject_Paper;
                MoveL target_aInf1Centro, v100, fine, tcptool\WObj:=Workobject_Paper;

	        ELSE

	        ENDIF
       ELSEIF "Fancy" = text_FontType THEN



	   ENDIF
    ENDPROC
ENDMODULE

--- Backups/Robot_ISEP_IRB140/RAPID/TASK1/PROGMOD/MainModule.mod ---
MODULE MainModule

        CONST robtarget Target_10:=[[0,0,0],[1,0,0,0],[0,-1,-2,0],[9E+09,9E+09,9E+09,9E+09,9E+09,9E+09]];
    CONST robtarget Target_20:=[[70,30,0],[1,0,0,0],[0,-1,-2,0],[9E+09,9E+09,9E+09,9E+09,9E+09,9E+09]];
    CONST robtarget Target_30:=[[0,60,0],[1,0,0,0],[0,-1,-2,0],[9E+09,9E+09,9E+09,9E+09,9E+09,9E+09]];
PROC main()
       ! Default sequence to reposition the robot
       startDefault;

       ! Main loop
        WHILE TRUE DO
            mainMenu;
        ENDWHILE


    ENDPROC
    PROC Path_A()
    ENDPROC
ENDMODULE

--- Backups/Robot_ISEP_IRB140/RAPID/TASK1/PROGMOD/Math.mod ---
MODULE Math
    ! ============== Declara??o de Variaveis =======================

    ! Apoio para as perguntas
    VAR num answer_impress;

    ! Write array
    PERS string char_impress;

    VAR num userInputTextLenght := 0;
    VAR num workSpaceWidth;
    VAR num workSpaceLength;
    VAR num letterLenghtAutomated;
    VAR num letterWidthAutomated;
    VAR num text_SpaceLettersAutomated;

    CONST num factorSpaceBetweenLetters := 5;
    CONST num factorHightLetter := 2;

    ! Position text
    VAR num xAvailable := 0 ;
    VAR num yAvailable := 0 ;
    VAR num coord_x_letter;
    VAR num coord_y_letter;

    PROC write_string()
        TPWrite "Insira a(s) palavra(s) pretendida(s) para imprimir.";
        userInputText := UIAlphaEntry(
            \Header:= "Impressão",
            \Message:= ""
            \Icon:=iconInfo
            \InitString:= "OPEN ROBOTICA");
    ENDPROC


    PROC calculateSizeLetterAutomated()
        ! Get the amount of chars in the array of text
        userInputTextLenght := StrLen(userInputText);

        ! Garentee the user actually inserts a text
        IF 0 = userInputTextLenght THEN
              TPWrite "Error : Necessário texto para poder imprimir.";
              errorA := TRUE;
              RETURN ;
        ENDIF

        ! Get the size of the page
        workSpaceWidth := paper_Width - paper_LeftMargin - paper_RightMargin ;
        workSpaceLength := paper_Length - paper_TopMargin - paper_BottomMargin ;

        ! Calculate the width of the text acordingly to fit the page line
        letterWidthAutomated := ( workSpaceWidth - ( ( userInputTextLenght - 1 ) * text_SpaceLetters ) ) DIV userInputTextLenght ;

        FOR I FROM 1 TO 10 DO
            ! Calculate the space required between letters
            text_SpaceLettersAutomated := text_SpaceLetters + letterWidthAutomated DIV factorSpaceBetweenLetters ;

            ! Recalculate the lenght of the text acordingly to fit the page line considering the new spacement
            letterWidthAutomated := ( workSpaceWidth - ( ( userInputTextLenght - 1 ) * text_SpaceLettersAutomated ) ) DIV userInputTextLenght ;
        ENDFOR

        ! Garantee a minimum space between
        IF 0 = text_SpaceLettersAutomated THEN
             text_SpaceLettersAutomated := 0.1;
        ENDIF

        ! Calcule the necessary height of letter
        letterLenghtAutomated := letterWidthAutomated * factorHightLetter;

        IF workSpaceLength  < letterLenghtAutomated  THEN
            letterLenghtAutomated := workSpaceLength ;
        ENDIF
    ENDPROC

    PROC calculateSizeLetterManual()
        ! Get the amount of chars in the array of text
        userInputTextLenght := StrLen(userInputText);

        ! Garentee the user actually inserts a text
        IF 0 = userInputTextLenght THEN
              TPWrite "Error : Necessário texto para poder imprimir.";
              errorA := TRUE;
              RETURN ;
        ENDIF

        ! Get the size of the page
        workSpaceWidth := paper_Width - paper_LeftMargin - paper_RightMargin ;
        workSpaceLength := paper_Length - paper_TopMargin - paper_BottomMargin ;

        ! Garantee a minimum space between
        IF 0 = text_SpaceLetters THEN
             text_SpaceLettersAutomated := 0.1;
        ENDIF
    ENDPROC

    PROC calculateOrigin( )
        IF FALSE = automatic THEN
	        IF "Esquerda" = paper_alignment THEN
	        	xAvailable := paper_LeftMargin;
	        ELSEIF "Direita" = paper_alignment THEN
	        	xAvailable := (workSpaceWidth) - ( letter_width * userInputTextLenght + userInputTextLenght * text_SpaceLetters ) ;
	        ELSEIF "Centrado" = paper_alignment THEN
	            xAvailable :=  paper_LeftMargin ;
	        ELSEIF "Justificado" = paper_alignment THEN
	        	xAvailable := paper_LeftMargin;
	        ENDIF

	        IF 0 = yAvailable THEN
	            yAvailable := paper_Length - paper_TopMargin - letter_lenght;
	        ELSE
	            yAvailable := coord_y_letter - letter_lenght - text_SpaceParag ;
	            !Condition to out page
	            IF 0 > yAvailable THEN
                     TPWrite "Error : Fora de página";
                     errorA := TRUE;

                    TPReadFK answerPaperMenu2,
                             stEmpty ,
                             "Nova Página" ,
                             "Ignorar" ,
                             stEmpty ,
                             stEmpty ,
                             "Voltar" ;

                    IF 1 = answerPaperMenu2 THEN
                       yAvailable := 0;
                    ENDIF
                    RETURN;
	            ENDIF
	        ENDIF


        ELSEIF TRUE = automatic THEN
	       	xAvailable := paper_LeftMargin;
	        IF 0 = yAvailable THEN
	            yAvailable := paper_Length - paper_TopMargin - letterLenghtAutomated;
	        ELSE
	            yAvailable := coord_y_letter - letterLenghtAutomated - text_SpaceParag ;
	            !Condition to out page
	            IF 0 > yAvailable THEN
                     TPWrite "Error : Fora de página";
                     errorA := TRUE;

                    TPReadFK answerPaperMenu2,
                             stEmpty ,
                             "Nova Página" ,
                             "Ignorar" ,
                             stEmpty ,
                             stEmpty ,
                             "Voltar" ;

                    IF 1 = answerPaperMenu2 THEN
                       yAvailable := 0;
                    ENDIF
                     RETURN;
	            ENDIF
	        ENDIF
        ENDIF

        coord_x_letter := xAvailable;
        coord_y_letter := yAvailable;
    ENDPROC
ENDMODULE

--- Backups/Robot_ISEP_IRB140/RAPID/TASK1/PROGMOD/Menu.mod ---
MODULE Menu

    ! ============== Definition of variables/constants =============================== !

    ! Questions suport
    VAR num answerInitMenu;
    VAR num answerPaperMenu;
    VAR num answerPaperMenu2;
    VAR num answerSettingMenu;
    VAR num answerWriteTextMenu;
    VAR num answerWriteTextMenu2;
    VAR num answerWrittingMenu;
    VAR num answerPrintingMenu;
    VAR num answerDebugMenu;

    ! Variable that stores the text input
    VAR string userInputText ;
    VAR string character;

    ! Dimensions of the format papers (mm)
    CONST num a3Lenght := 297;
    CONST num a3Width := 420;
    CONST num a4Lenght := 210;
    CONST num a4Width := 297;
    CONST num a5Lenght := 148;
    CONST num a5Width := 210;

    ! Initialize the paper characteristics
    VAR string paper_size := "A4";
    VAR string paper_orientation := "Vertical";
    VAR string paper_alignment := "Esquerda";
    VAR num paper_TopMargin := 20;
    VAR num paper_BottomMargin := 20;
    VAR num paper_LeftMargin := 10;
    VAR num paper_RightMargin := 10;
    VAR num paper_Width := a4Lenght;
    VAR num paper_Length := a4Width;

    ! Initialize the text characteristics
    VAR string text_FontType := "Classic";
    VAR num text_SizePT := 12;
    VAR string text_Color := "Black";
    VAR num text_Rotation := 0;
    VAR num text_SpaceLetters := 2;
    VAR num text_SpaceParag := 5;

    ! Initialize letters characteristics
    VAR num letter_lenght := 5;
    VAR num letter_width := 10;

    VAR num paragraph_write := 0;

    VAR bool automatic := FALSE;

    VAR num altura_letras;
    VAR num comprimento_letras;

    VAR bool errorA := FALSE;

    VAR iodev file;

    ! ==================== Code - default ========================= !

    ! Process for the inicialization program
    PROC startDefault( )
        ! Clear console
        TPErase;

        MoveJ Default_position,v1000,fine,tcptool\WObj:=Workobject_Paper;

        ! JumpHome; !TODO
        TPWrite "O robot está pronto a ser operado.";

        WaitTime(1);
    ENDPROC

    ! ==================== Code - mainMenu ======================== !

    PROC mainMenu()
        !Clear console
        TPErase;

        ! Welcome page.
        TPWrite "Plotter & Open Robótica";

        ! Options of the menu
        TPReadFK answerInitMenu ,
                 stEmpty ,
                 "Escrever Manualmente" ,
                 "Definições texto" ,
                 "Definições folha" ,
                 "Imprimir",
                 "Debug";

        IF 1 = answerInitMenu THEN
            writeTextMenu;
        ELSEIF 2 = answerInitMenu THEN
           answersettingMenu := 0;
           settingsTextMenu ;
        ELSEIF 3 = answerInitMenu THEN
            settingsPageMenu ;
        ELSEIF 4 = answerInitMenu THEN
            printingPageMenu ;
        ELSEIF 5 = answerInitMenu THEN
            debugMenu ;
        ENDIF
    ENDPROC

    ! ==================== Code - writeMenu ======================= !

    PROC writeTextMenu( )
        WHILE answerWrittingMenu <> 5 DO
            ! Clear the console
            TPErase;

            TPWrite("Frase a escrever:");
            ! Options to change settings of the page
            TPReadFK answerSettingMenu,
                     userInputText ,
                     "Escrever",
                     "Gerar Nova Página",
                     stEmpty,
                     stEmpty,
                     "Voltar";

            IF 1 = answersettingMenu THEN
                write_string;

            ELSEIF 2 = answersettingMenu THEN
                yAvailable := 0;

            ELSEIF 3 = answersettingMenu THEN

            ELSEIF 4 = answersettingMenu THEN

            ELSEIF 5 = answersettingMenu THEN
                answerWrittingMenu := 5;
                ! Back to menu
            ENDIF
        ENDWHILE
        answerWrittingMenu := 0;
    ENDPROC

    ! ==================== Code - settingsText ==================== !

    PROC settingsTextMenu( )
        WHILE answersettingMenu <> 5 DO
            ! Clear the console
            TPErase;

            tpWriteReportSettingsTextMenu;

            ! Options to change settings of the page
            TPReadFK answerSettingMenu,
                     stEmpty ,
                     "Fonte",
                     "Tamanho (pt)",
                     "Cor",
                     "Página seguinte",
                     "Voltar";

            IF 1 = answersettingMenu THEN
                fontTypePageMenu ;

            ELSEIF 2 = answersettingMenu THEN
                TPReadNum text_SizePT, "Qual é o tamanho da letra? (pt) (default = 12)";
                !TODO convert pt to mm

            ELSEIF 3 = answersettingMenu THEN
                fontColorPageMenu ;

            ELSEIF 4 = answersettingMenu THEN
                answersettingMenu := 0;
                settingsTextMenu2 ;

            ELSEIF 5 = answersettingMenu THEN
                answersettingMenu := 5;
                ! Back to menu
            ENDIF

        ENDWHILE
    ENDPROC

    PROC settingsTextMenu2( )
        WHILE answersettingMenu <> 5 DO
            ! Clear the console
            TPErase;

            tpWriteReportSettingsTextMenu;

            ! Options to change settings of the page
            TPReadFK answerSettingMenu,
                     stEmpty ,
                     "Rotação",
                     "Espaçamento entre letras",
                     "Espaçamento entre paragráfos",
                     "Página seguinte",
                     "Voltar";

            IF 1 = answersettingMenu THEN
                TPReadNum text_Rotation, "Qual é a rotação pretendida? (graus)";

            ELSEIF 2 = answersettingMenu THEN
                TPReadNum text_SpaceLetters, "Qual é o espaçamento entre letras? (mm) (default = 2)";

            ELSEIF 3 = answersettingMenu THEN
                TPReadNum text_SpaceParag, "Qual é o espaçamento entre paragráfos? (mm) (default = 5)";

            ELSEIF 4 = answersettingMenu THEN
                answersettingMenu := 0;
                settingsTextMenu3 ;

            ELSEIF 5 = answersettingMenu THEN
                answersettingMenu := 5;
                ! Back to menu
            ENDIF
        ENDWHILE
    ENDPROC

    PROC settingsTextMenu3( )
        WHILE answersettingMenu <> 5 DO
            ! Clear the console
            TPErase;

            tpWriteReportSettingsTextMenu;

            ! Options to change settings of the page
            TPReadFK answerSettingMenu,
                     stEmpty ,
                     "Negrito",
                     "Itálico",
                     "Sublinhado",
                     "Página seguinte",
                     "Voltar";

            IF 1 = answersettingMenu THEN
                 ! Do nothing yet

            ELSEIF 2 = answersettingMenu THEN
                 ! Do nothing yet

            ELSEIF 3 = answersettingMenu THEN
                 ! Do nothing yet

            ELSEIF 4 = answersettingMenu THEN
                answersettingMenu := 0;
                settingsTextMenu ;
            ELSEIF 5 = answersettingMenu THEN
                answersettingMenu := 5;
                ! Back to menu
            ENDIF
        ENDWHILE
    ENDPROC


    PROC tpWriteReportSettingsTextMenu()
        ! Clear the console
        TPErase;

        TPWrite("Definições de Texto:");

        ! Display font type
        TPWrite("Fonte de Letra: " + text_FontType );

        ! Display letter size
        TPWrite "Tamanho de letra:" + NumToStr(text_SizePT,0) + "pt" + "(" + NumToStr(letter_lenght,0) + " mm , " +  NumToStr(letter_width,0) + " mm )";

        ! Display letter color
        TPWrite "Cor de Letra: " + text_Color;

        ! Display letter rotation
        TPWrite "Rotação do texto: " + NumToStr( text_Rotation, 0 ) + " graus";

        ! Display space between letters
        TPWrite "Espaçamento entre letras: " + NumToStr( text_SpaceLetters, 0 ) + " mm";

        ! Display space between paragraphs
        TPWrite "Espaçamento entre parágrafos: " + NumToStr( text_SpaceParag, 0 ) + " mm";
    ENDPROC

    PROC fontTypePageMenu( )
        ! Clear the console
        TPErase;

        tpWriteReportSettingsTextMenu;

        ! Options to change format
        TPReadFK answerWriteTextMenu2,
                 stEmpty ,
                 "Classic" ,
                 "Digital" ,
                 "Fancy" ,
                 stEmpty ,
                 "Voltar" ;

        IF 1 = answerWriteTextMenu2 THEN
            text_FontType := "Classic";

        ELSEIF 2 = answerWriteTextMenu2 THEN
            text_FontType := "Digital";

        ELSEIF 3 = answerWriteTextMenu2 THEN
            text_FontType := "Fancy";

        ELSEIF 4 = answerWriteTextMenu2 THEN
            ! nothing for now (fuction enable)

        ELSEIF 5 = answerWriteTextMenu2 THEN
            answerWriteTextMenu2 := 0 ;
        ENDIF
    ENDPROC

    PROC fontColorPageMenu( )
        ! Clear the console
        TPErase;

        tpWriteReportSettingsTextMenu;

        ! Options to change format
        TPReadFK answerWriteTextMenu2,
                 stEmpty ,
                 "Preto" ,
                 "Azul" ,
                 "Vermelho" ,
                 stEmpty ,
                 "Voltar" ;

        IF 1 = answerWriteTextMenu2 THEN
            text_Color := "Black";

        ELSEIF 2 = answerWriteTextMenu2 THEN
            text_Color := "Blue";

        ELSEIF 3 = answerWriteTextMenu2 THEN
            text_Color := "Red";

        ELSEIF 4 = answerWriteTextMenu2 THEN
            ! nothing for now (fuction enable)

        ELSEIF 5 = answerWriteTextMenu2 THEN
            answerWriteTextMenu2 := 0 ;
        ENDIF
    ENDPROC


    ! ==================== Code - settingsPage ==================== !

    PROC settingsPageMenu( )
        WHILE 5 <> answerPaperMenu DO
            ! Clear the console
            TPErase;

            tpWriteReportSettingsPageMenu;

            ! Options to change settings of the page
            TPReadFK answerPaperMenu,
                     stEmpty ,
                     "Formato",
                     "Orientação",
                     "Margens",
                     "Alinhamento",
                     "Voltar";

            IF 1 = answerPaperMenu THEN
                formatPageMenu ;
                yAvailable := 0;

            ELSEIF 2 = answerPaperMenu THEN
                orientationPageMenu;
                yAvailable := 0;

            ELSEIF 3 = answerPaperMenu THEN
                marginsPageMenu ;

            ELSEIF 4 = answerPaperMenu THEN
                alignmentPageMenu ;

            ELSEIF 5 = answerPaperMenu THEN !Go out in the while
            ENDIF
        ENDWHILE

        answerPaperMenu := 0;
    ENDPROC

    PROC tpWriteReportSettingsPageMenu()
        TPWrite("Definições de página:");

        ! Display paper size
        TPWrite "Formato da folha: " + paper_size + " ( " +  NumToStr(paper_Width,0) + " mm, " +  NumToStr(paper_Length,0) + " mm)";

        ! Display paper orientation
        TPWrite "Orientação da folha: " + paper_Orientation;

        ! Display paper margins
        TPWrite "Margens da folha: ";
        TPWrite " " + NumToStr( paper_TopMargin, 0 ) + " (mm) (cabeçalho)," + NumToStr( paper_BottomMargin ,0 ) + " (mm) (rodapé)," ;
        TPWrite " " + NumToStr( paper_LeftMargin, 0 ) + " (mm) (esquerda)," + NumToStr( paper_RightMargin , 0 ) + " (mm) (direita)" ;

        ! Display text alignment
        TPWrite("Alinhamento do texto: " + paper_Alignment );
    ENDPROC

    PROC formatPageMenu( )
        ! Clear the console
        TPErase;

        tpWriteReportSettingsPageMenu;

        ! Options to change format
        TPReadFK answerPaperMenu2,
                 stEmpty ,
                 "A3" ,
                 "A4" ,
                 "A5" ,
                 stEmpty ,
                 "Voltar" ;

        IF 1 = answerPaperMenu2 THEN
            paper_size := "A3" ;

            IF "Vertical" = paper_orientation THEN
                 paper_Width := a3Lenght;
                 paper_Length := a3Width;
            ELSE
                 paper_Width := a3Width;
                 paper_Length := a3Lenght;
            ENDIF

        ELSEIF 2 = answerPaperMenu2 THEN
            paper_size := "A4" ;

            IF "Vertical" = paper_orientation THEN
                 paper_Width := a4Lenght;
                 paper_Length := a4Width;
            ELSE
                 paper_Width := a4Width;
                 paper_Length := a4Lenght;
            ENDIF

        ELSEIF 3 = answerPaperMenu2 THEN
            paper_size := "A5" ;

            IF "Vertical" = paper_orientation THEN
                 paper_Width := a5Lenght;
                 paper_Length := a5Width;
            ELSE
                 paper_Width := a5Width;
                 paper_Length := a5Lenght;
            ENDIF

        ELSEIF 4 = answerPaperMenu2 THEN
            ! nothing for now (fuction enable)

        ELSEIF 5 = answerPaperMenu2 THEN
            answerPaperMenu2 := 0 ;
        ENDIF
    ENDPROC

    PROC orientationPageMenu( )
        ! Clear the console
        TPErase;

        tpWriteReportSettingsPageMenu;

        ! Options to change orientation
        TPReadFK answerPaperMenu2,
                 stEmpty ,
                 "Horizontal" ,
                 "Vertical" ,
                 stEmpty ,
                 stEmpty ,
                 "Voltar" ;

        IF 1 = answerPaperMenu2 THEN
            paper_Orientation := "Horizontal";
            IF paper_size = "A3" THEN
                paper_Width := a3Width;
                paper_Length := a3Lenght;
            ELSEIF paper_size = "A4" THEN
                paper_Width := a4Width;
                paper_Length := a4Lenght;
            ELSEIF paper_size = "A5" THEN
                paper_Width := a5Width;
                paper_Length := a5Lenght;
            ENDIF

        ELSEIF 2 = answerPaperMenu2 THEN
            paper_Orientation := "Vertical";
            IF paper_size = "A3" THEN
                paper_Width := a3Lenght;
                paper_Length := a3Width;
            ELSEIF paper_size = "A4" THEN
                paper_Width := a4Lenght;
                paper_Length := a4Width;
            ELSEIF paper_size = "A5" THEN
                paper_Width := a5Lenght;
                paper_Length := a5Width;
            ENDIF

        ELSEIF 3 = answerPaperMenu2 THEN
            ! nothing for now

        ELSEIF 4 = answerPaperMenu2 THEN
            ! nothing for now

        ELSEIF 5 = answerPaperMenu2 THEN
            answerPaperMenu2 := 0 ;
        ENDIF
    ENDPROC

    PROC marginsPageMenu( )
        ! Clear the console
        TPErase;

        tpWriteReportSettingsPageMenu;

        ! Options to change orientation
        TPReadFK answerPaperMenu2,
                 stEmpty ,
                 "Cabeçalho" ,
                 "Rodapé" ,
                 "Direita" ,
                 "Esquerda" ,
                 "Voltar" ;

        ! TODO does nothing at the moment

        IF 1 = answerPaperMenu2 THEN
            TPReadNum paper_TopMargin, "Qual é o valor da margem do cabe alho? (mm)";

        ELSEIF 2 = answerPaperMenu2 THEN
            TPReadNum paper_BottomMargin, "Qual é o valor da margem do rodap ? (mm)";

        ELSEIF 3 = answerPaperMenu2 THEN
            TPReadNum paper_RightMargin, "Qual é o valor da margem direita? (mm)";

        ELSEIF 4 = answerPaperMenu2 THEN
            TPReadNum paper_LeftMargin, "Qual é o valor da margem esquerda? (mm)";

        ELSEIF 5 = answerPaperMenu2 THEN
            answerPaperMenu2 := 0 ;
        ENDIF
    ENDPROC

    PROC alignmentPageMenu( )
        ! Clear the console
        TPErase;

        tpWriteReportSettingsPageMenu;

        ! Options to change orientation
        TPReadFK answerPaperMenu2,
                 stEmpty ,
                 "Centro" ,
                 "Esquerda" ,
                 "Direita" ,
                 "Justificado" ,
                 "Voltar" ;

        IF 1 = answerPaperMenu2 THEN
            paper_Alignment := "Centro";

        ELSEIF 2 = answerPaperMenu2 THEN
            paper_Alignment := "Esquerda";

        ELSEIF 3 = answerPaperMenu2 THEN
            paper_Alignment := "Direita";

        ELSEIF 4 = answerPaperMenu2 THEN
            paper_Alignment := "Justificado";

        ELSEIF 5 = answerPaperMenu2 THEN
            answerPaperMenu2 := 0 ;
        ENDIF
    ENDPROC


    !===================== Code - ImpressMenu ============================

    PROC printingPageMenu()
         VAR num x := 1;
        WHILE answerPrintingMenu = 4 OR answerPrintingMenu = 0 DO
           ! Clear the console
           TPErase;

           IF 1 = x THEN
                TPWrite "Texto a ser impresso";
                TPWrite userInputText;
    	        x := 2;
            ELSEIF 2 = X THEN
	            tpWriteReportSettingsTextMenu;
    	        x := 3;
            ELSE
                tpWriteReportSettingsPageMenu;
    	        x := 1;
            ENDIF

            ! Options to change settings of the page
            TPReadFK answerPrintingMenu,
                     stEmpty ,
                     "Automático",
                     "Manual",
                     "Ficheiro",
                     "Scroll",
                     "Voltar";

            IF 1 = answerPrintingMenu THEN
                automatic := TRUE;
                calculateSizeLetterAutomated;
                calculateOrigin;
                IF TRUE = errorA THEN
                    automatic := FALSE;
                    errorA := FALSE;
                    RETURN;
                ENDIF

                altura_letras := letterLenghtAutomated ;
                comprimento_letras := letterWidthAutomated ;

                impressMecanism;
                automatic := FALSE;

            ELSEIF 2 = answerPrintingMenu THEN
                manualPriting;
            ELSEIF 3 = answerPrintingMenu THEN
                Open "HOME:"\File:="file.txt", file, \Read;
                userInputText := "";
                WHILE userInputText <> "EOF" DO
                    IF userInputText <> EOF THEN
                        userInputText := ReadStr(file, \Delim:=";");
                        manualPriting;
                        ! ITS IMPRESSING EOF
                    ENDIF
                ENDWHILE
	            Close file;
            ELSEIF 4 = answerPrintingMenu THEN


            ELSEIF 5 = answerPrintingMenu THEN
                answerPrintingMenu := 5;
                ! Back to menu
            ENDIF
        ENDWHILE
        answerPrintingMenu := 0;
    ENDPROC


    PROC manualPriting()
        automatic := FALSE;
        calculateSizeLetterManual;

        letter_width := text_SizePT * 0.35;
        letter_lenght := letter_width * factorHightLetter;
        altura_letras := letter_lenght ;
        comprimento_letras := letter_width ;

        calculateOrigin;
        IF TRUE = errorA THEN
            automatic := FALSE;
            errorA := FALSE;
            RETURN;
        ENDIF


        impressMecanism;
    ENDPROC

    ! ==================== Code - debugMenu ==================== !

    PROC debugMenu( )
        ! Clear the console
        TPErase;


        ! Options to change settings of the page
            TPReadFK answerDebugMenu,
                     "Menu de depuração" ,
                     "Alfabeto",
                     "WorkObj",
                     "Offset Z",
                     Stempty,
                     "Voltar";

            IF 1 = answerDebugMenu THEN
                userInputText := "ABCDEFGHIJKLMNOPQRSTUVWXYZ 0123456789";
            ELSEIF 2 = answerDebugMenu THEN
                workobjectSelector;

            ELSEIF 3 = answerDebugMenu THEN
                TPReadNum offsetZo, "CUIDADO: Qual é o offset em Z? (mm)";

            ELSEIF 4 = answerDebugMenu THEN

            ELSEIF 5 = answerDebugMenu THEN
                answerDebugMenu := 0;
                ! Back to menu
            ENDIF

        !TPRead
    ENDPROC

    PROC workobjectSelector()
        ! Clear the console
        TPErase;


        ! Options to change settings of the page
        TPReadFK answerDebugMenu,
                 "Escolha de workobject" ,
                 "A3",
                 "A4",
                 "A5",
                 Stempty,
                 "Voltar";

        IF 1 = answerDebugMenu THEN

        ELSEIF 2 = answerDebugMenu THEN
              Workobject_Paper := WA4;

        ELSEIF 3 = answerDebugMenu THEN
              Workobject_Paper := WA5;

        ELSEIF 4 = answerDebugMenu THEN

        ELSEIF 5 = answerDebugMenu THEN
            answerDebugMenu := 0;
            ! Back to menu
        ENDIF
    ENDPROC
ENDMODULE

--- Backups/Robot_ISEP_IRB140/RAPID/TASK1/PROGMOD/Module1.mod ---
MODULE Module1
    PROC Path_Start()

    ENDPROC
    PROC Path_10()
        MoveL Default_position,v1000,z100,pen\WObj:=Workobject_Paper;
        MoveL Origem,v1000,z100,pen\WObj:=Workobject_Paper;
    ENDPROC
ENDMODULE

--- Backups/Robot_ISEP_IRB140/RAPID/TASK1/PROGMOD/Print.mod ---
MODULE Print
    CONST num time := 1;

    PROC impressMecanism()
        TPErase;
        !TPWrite NumtoStr(coord_y_letter,0);
        TPWrite "A imprimir  ...";

		FOR i FROM 1 TO StrLen( userInputText ) DO
            character := StrPart( userInputText, i, 1);
            draw;

            !TPWrite NumToStr(coord_x_letter,0);
            !WaitTime(2);
            !Calculate new point center

            IF TRUE = automatic THEN
                coord_x_letter := coord_x_letter + letterWidthAutomated + text_SpaceLettersAutomated ;
            ELSE
               coord_x_letter := coord_x_letter + letter_width + text_SpaceLetters;
               IF (coord_x_letter + letter_width) > workSpaceWidth THEN
                     calculateOrigin;
               ENDIF
            ENDIF
		ENDFOR

        TPWrite "Impressão Feita";

        MoveJ Default_position, v100 , fine , tcptool\WObj:=Workobject_Paper ;
        WaitTime( time );
    ENDPROC
    PROC impress_mecanism()
        draw;
        MoveJ Default_position,v1000,fine,tcptool\WObj:=Workobject_Paper;
        WaitTime( time );
    ENDPROC
ENDMODULE

--- Backups/Robo_open_v2/RAPID/TASK0/SYSMOD/guisocks.sys ---
module guisocks(sysmodule)

   pers num nGUISockCmdId    := 0;
   pers num nGUISockClientId := 0;
   pers num nGUISockSerNo    := 0;

   pers num nGUISockPars{10}      := [0,0,0,0,0,0,0,0,0,0];
   pers string stGUISockPar{1}    := [""];
   pers num nGUISockRetPars{10}   := [0,0,0,0,0,0,0,0,0,0];
   pers string stGUISockRetPar{1} := [""];

endmodule

--- Backups/Robo_open_v2/RAPID/TASK0/SYSMOD/pntcmds.sys ---
module pntcmds(sysmodule)
   !
   ! (C) Copyright 2007 ABB
   !



   pers num nIntCommand          := 0;
   pers num nIntInParams{10}     := [0,0,0,0,0,0,0,0,0,0];
   pers string stIntInParams{1}  := [""];
   pers num nIntOutParams{10}    := [0,0,0,0,0,0,0,0,0,0];
   pers string stIntOutParams{1} := [""];



endmodule

--- Backups/Robo_open_v2/RAPID/TASK0/SYSMOD/syselog.sys ---
module syselog(sysmodule)

   !
   ! (C) Copyright 2005 ABB
   !
   const num PNT_ELOG_INFO    := 1;
   const num PNT_ELOG_WARNING := 2;
   const num PNT_ELOG_ERROR   := 3;

   proc PntElog(
      num elog_number,
      num type_err,
      \string Arg1,
      \string Arg2,
      \string Arg3,
      \string Arg4,
      \string Arg5)

      ! SysFun1. Undocumented hidden function.
      ! Scope: Used to write internal messages in common/process elog.
      ! This function shall NOT be used by our customers.
      ! Type_err :
      !           1 = Information
      !           2 = Warning
      !           3 = Error

      const num domain_no := 13;
      var string stArg1 := ERRSTR_UNUSED;
      var string stArg2 := ERRSTR_UNUSED;
      var string stArg3 := ERRSTR_UNUSED;
      var string stArg4 := ERRSTR_UNUSED;
      var string stArg5 := ERRSTR_UNUSED;


      if Present(Arg1) stArg1 := Arg1;
      if Present(Arg2) stArg2 := Arg2;
      if Present(Arg3) stArg3 := Arg3;
      if Present(Arg4) stArg4 := Arg4;
      if Present(Arg5) stArg5 := Arg5;

      SysFun1
         domain_no,
         elog_number,
         type_err ,
         stArg1,
         stArg2,
         stArg3,
         stArg4,
         stArg5;
   error
      Break; ! Unhandled error.
   endproc

endmodule

--- Backups/Robo_open_v2/RAPID/TASK0/SYSMOD/tpusocks.sys ---
module tpusocks(sysmodule)

   pers num nTPUSockCmdId    := 0;
   pers num nTPUSockClientId := 0;
   pers num nTPUSockSerNo    := 0;

   pers num nTPUSockPars{10}      := [0,0,0,0,0,0,0,0,0,0];
   pers string stTPUSockPar{1}    := [""];
   pers num nTPUSockRetPars{10}   := [0,0,0,0,0,0,0,0,0,0];
   pers string stTPUSockRetPar{1} := [""];

endmodule

--- Backups/Robo_open_v2/RAPID/TASK1/SYSMOD/bfdata.sys ---
module bfdata(sysmodule)



   const num BF_FLUID_CHANNEL := 1;
   const num BF_APPLICATORS := 1;
   const num BF_CHANNELS := 5;
   const num BF_MATERIALS := 100;

   pers bool bImmediateFactor := true; ! Indicate if also set immediately.
   pers bool bSkipBrushFactor; ! Set for each cycle as needed.

   pers num nCurrentFactor{BF_APPLICATORS, BF_CHANNELS} :=
     [[100,100,100,100,100]]; ! Current factors used for the current job.

   pers num nGlobalFactor{BF_APPLICATORS, BF_CHANNELS} :=
     [[100,100,100,100,100]];

   pers num nMaterialFactor{BF_MATERIALS, BF_APPLICATORS, BF_CHANNELS} :=
    [[[100,100,100,100,100]],
     [[100,100,100,100,100]],
     [[100,100,100,100,100]],
     [[100,100,100,100,100]],
     [[100,100,100,100,100]],
     [[100,100,100,100,100]],
     [[100,100,100,100,100]],
     [[100,100,100,100,100]],
     [[100,100,100,100,100]],
     [[100,100,100,100,100]],
     [[100,100,100,100,100]],
     [[100,100,100,100,100]],
     [[100,100,100,100,100]],
     [[100,100,100,100,100]],
     [[100,100,100,100,100]],
     [[100,100,100,100,100]],
     [[100,100,100,100,100]],
     [[100,100,100,100,100]],
     [[100,100,100,100,100]],
     [[100,100,100,100,100]],
     [[100,100,100,100,100]],
     [[100,100,100,100,100]],
     [[100,100,100,100,100]],
     [[100,100,100,100,100]],
     [[100,100,100,100,100]],
     [[100,100,100,100,100]],
     [[100,100,100,100,100]],
     [[100,100,100,100,100]],
     [[100,100,100,100,100]],
     [[100,100,100,100,100]],
     [[100,100,100,100,100]],
     [[100,100,100,100,100]],
     [[100,100,100,100,100]],
     [[100,100,100,100,100]],
     [[100,100,100,100,100]],
     [[100,100,100,100,100]],
     [[100,100,100,100,100]],
     [[100,100,100,100,100]],
     [[100,100,100,100,100]],
     [[100,100,100,100,100]],
     [[100,100,100,100,100]],
     [[100,100,100,100,100]],
     [[100,100,100,100,100]],
     [[100,100,100,100,100]],
     [[100,100,100,100,100]],
     [[100,100,100,100,100]],
     [[100,100,100,100,100]],
     [[100,100,100,100,100]],
     [[100,100,100,100,100]],
     [[100,100,100,100,100]],
     [[100,100,100,100,100]],
     [[100,100,100,100,100]],
     [[100,100,100,100,100]],
     [[100,100,100,100,100]],
     [[100,100,100,100,100]],
     [[100,100,100,100,100]],
     [[100,100,100,100,100]],
     [[100,100,100,100,100]],
     [[100,100,100,100,100]],
     [[100,100,100,100,100]],
     [[100,100,100,100,100]],
     [[100,100,100,100,100]],
     [[100,100,100,100,100]],
     [[100,100,100,100,100]],
     [[100,100,100,100,100]],
     [[100,100,100,100,100]],
     [[100,100,100,100,100]],
     [[100,100,100,100,100]],
     [[100,100,100,100,100]],
     [[100,100,100,100,100]],
     [[100,100,100,100,100]],
     [[100,100,100,100,100]],
     [[100,100,100,100,100]],
     [[100,100,100,100,100]],
     [[100,100,100,100,100]],
     [[100,100,100,100,100]],
     [[100,100,100,100,100]],
     [[100,100,100,100,100]],
     [[100,100,100,100,100]],
     [[100,100,100,100,100]],
     [[100,100,100,100,100]],
     [[100,100,100,100,100]],
     [[100,100,100,100,100]],
     [[100,100,100,100,100]],
     [[100,100,100,100,100]],
     [[100,100,100,100,100]],
     [[100,100,100,100,100]],
     [[100,100,100,100,100]],
     [[100,100,100,100,100]],
     [[100,100,100,100,100]],
     [[100,100,100,100,100]],
     [[100,100,100,100,100]],
     [[100,100,100,100,100]],
     [[100,100,100,100,100]],
     [[100,100,100,100,100]],
     [[100,100,100,100,100]],
     [[100,100,100,100,100]],
     [[100,100,100,100,100]],
     [[100,100,100,100,100]],
     [[100,100,100,100,100]]];



     ! Helper function to allow "late binding" setting of the value.
     proc ImmediateFactor(bool bValue)
        bImmediateFactor := bValue;
     endproc



     ! Calculate actual volume to be used with the factor applied.
     proc RetrFactorComp(inout num nVolume, num nMaterial, num nApp)
        nVolume := nVolume *
                  (nGlobalFactor{nApp, BF_FLUID_CHANNEL} / 100) *
                  (nMaterialFactor{nMaterial, nApp, BF_FLUID_CHANNEL} / 100);
     endproc



     ! Calculate real volume to store (100% factor) with the factor applied.
     ! Must use currently used factor for the job, in case it was changed while painting!
     proc StoreFactorComp(inout num nVolume, num nApp)
        nVolume := nVolume / (nCurrentFactor{nAPP, BF_FLUID_CHANNEL} / 100);
     endproc



endmodule

--- Backups/Robo_open_v2/RAPID/TASK1/SYSMOD/config.sys ---
module config(sysmodule)



   local const num MAX_OPTIONS := 20;
   local const num MAX_AREA := 5;

   pers string stOptionNames{MAX_AREA, MAX_OPTIONS};
   pers string stOptionValues{MAX_AREA, MAX_OPTIONS};
   pers string stAreaMapping{MAX_AREA};
   pers stringdig sdAreaFileTimes{MAX_AREA} := ["1710267316", "0", "0", "0", "0"];

   pers bool bConfigSemaphore;



   local func num nAreaMap(string stArea)
      for i from 1 to Dim(stAreaMapping, 1) do
         if stArea = stAreaMapping{i}
            return i;
      endfor
      return 0;
   endfunc



   local func bool bNewAreaMap(string stArea)
      for i from 1 to Dim(stAreaMapping, 1) do
         if stAreaMapping{i} = "" then
            stAreaMapping{i} := stArea;
            return true;
         endif
      endfor
      return false;
   endfunc



   func string stPntRapidOption(string stArea, string stOption)
      var bool bDoReRead;
      var string stFilePath;
      var string stValue := "";
      var stringdig sdFileTime;
      var bool bTimeOut;

      WaitUntil TestAndSet(bConfigSemaphore) \MaxTime := 5 \TimeFlag := bTimeOut;
      if bTimeOut then
         PntElog 4068, PNT_ELOG_ERROR \Arg1 := stArea \Arg2 := stOption;
         bConfigSemaphore := false; ! To get out of a deadlock situation.
         return "";
      endif

      stFilePath := HOME_ROOT + stArea + ".xml";

      if nAreaMap(stArea) = 0 then
         ! Area not used before, create new mapping.
         if IsFile(stFilePath) then
            if not bNewAreaMap(stArea) then
               PntElog 4055, PNT_ELOG_ERROR \Arg1 := stArea \Arg2 := stOption;
               bConfigSemaphore := false;
               return "";
            endif
         else
            PntElog 4056, PNT_ELOG_ERROR \Arg1 := stArea \Arg2 := stOption;
            bConfigSemaphore := false;
            return "";
         endif
         bDoReRead := true;
      else
         if FileTime(stFilePath \ModifyTime, \StrDig := sdFileTime) > 0 and
            StrDigCmp(sdAreaFileTimes{nAreaMap(stArea)}, LT, sdFileTime) then
            sdAreaFileTimes{nAreaMap(stArea)} := sdFileTime;
            bDoReRead := true;
         else
            bDoReRead := false;
         endif
      endif

      if bDoReRead then
         if nParseXMLFile(stFilePath, stOptionNames, stOptionValues, nAreaMap(stArea)) = 0 then
            PntElog 4057, PNT_ELOG_ERROR \Arg1 := stArea \Arg2 := stOption;
            bConfigSemaphore := false;
            return "";
         endif
      endif

      bConfigSemaphore := false;

      for i from 1 to Dim(stOptionNames, 2) do
         ! Case in-sensitive compare.
         if StrMap(stOptionNames{nAreaMap(stArea), i}, STR_LOWER, STR_UPPER) =
            StrMap(stArea + "/" + stOption, STR_LOWER, STR_UPPER)
            stValue := stOptionValues{nAreaMap(stArea), i};
      endfor

      if stValue = ""
         PntElog 4058, PNT_ELOG_ERROR \Arg1 := stArea \Arg2 := stOption;

      return stValue;
   error
      if errno = ERR_FILEACC then
         ! File has been deleted for some reason.
         PntElog 4062, PNT_ELOG_ERROR \Arg1 := stFilePath;
         bConfigSemaphore := false;
         return "";
      endif
   endfunc



   func bool bIsTrue(string stStatement)
      var num nTemp;

      ! Accept "1" as true.
      if StrToVal(stStatement, nTemp) then
         if nTemp = 1
            return true;
      endif

      ! Accept case insensitive "True" as true.
      if StrMap(stStatement, STR_LOWER, STR_UPPER) = "TRUE"
         return true;

      ! Accept case insensitive "Yes" as true.
      if StrMap(stStatement, STR_LOWER, STR_UPPER) = "YES"
         return true;

      return false;
   endfunc



   ! Very simple XML parser with only one stack depth (called the area).
   local func num nParseXMLFile(string stFileName, inout string stNames{*,*}, inout string stValues{*,*}, num nFirstDimension)
      var iodev ioFile;
      var string stLine;
      var string stCurrentArea := "";
      var num nOptionCount := 1;

      if nFirstDimension > Dim(stNames, 1) or nFirstDimension > Dim(stValues, 1) then
         PntElog 4059, PNT_ELOG_ERROR;
         return 0;
      endif

      ! Options are saved as paths like "Kernel/LogEnable" as the first dimension.

      Open stFileName, ioFile \Read;
      while stLine <> EOF do
         stLine := ReadStr(ioFile \RemoveCR);
         if stLine <> EOF then
            if StrMatch(stLine, 1, "<?") < StrLen(stLine) then
               ! Skip the XML header.
            elseif StrFind(stLine, 1, "=") < StrLen(stLine) then
               ! Line contains equal sign, so it must be an option=value tag.
               if stCurrentArea <> "" then
                  stNames{nFirstDimension, nOptionCount} := stCurrentArea + "/" + stStringBetween(stLine, "<", " ");
               else
                  stNames{nFirstDimension, nOptionCount} := stStringBetween(stLine, "<", " ");
               endif
               stValues{nFirstDimension, nOptionCount} := stStringBetween(stLine, """", """");
               Incr nOptionCount;
               if nOptionCount > Dim(stNames, 2) or nOptionCount > Dim(stValues, 2) then
                  PntElog 4061, PNT_ELOG_ERROR \Arg1 := stFileName \Arg2 := ValToStr(nOptionCount - 1);
                  Close ioFile;
                  return nOptionCount - 1;
               endif
            else
               ! No equal sign means it must be an "area" tag.
               if StrFind(stLine, 1, "/") < StrLen(stLine) then
                  ! Containing slash means the "area" is finished.
                  stCurrentArea := "";
               else
                  ! No slash means start of new "area".
                  stCurrentArea := stStringBetween(stLine, "<", ">");
               endif
            endif
         endif
      endwhile
      Close ioFile;

      return nOptionCount - 1;
   error
      if errno = ERR_FILEOPEN then
         PntElog 4062, PNT_ELOG_ERROR \Arg1 := stFileName;
         return 0;
      endif
   endfunc



   local func string stStringBetween(string stString, string stStart, string stEnd)
      var num nStartPos;
      var num nEndPos;

      nStartPos := StrMatch(stString, 1, stStart);
      if nStartPos > StrLen(stString) then
         PntElog 4063, PNT_ELOG_ERROR;
         return "";
      endif

      nEndPos := StrMatch(stString, nStartPos + 1, stEnd);
      if nEndPos > StrLen(stString) then
         PntElog 4063, PNT_ELOG_ERROR;
         return "";
      endif

      return StrPart(stString, nStartPos + 1, (nEndPos - nStartPos - 1));
   endfunc



endmodule

--- Backups/Robo_open_v2/RAPID/TASK1/SYSMOD/constant.sys ---
module constant(sysmodule)
   !
   ! (C) Copyright 2007 ABB
   !



   ! Command results:
   const num CMD_OK          := 0;
   const num CMD_FAILED      := -1;
   const num CMD_UNKNOWN     := -2;
   const num CMD_NOT_MASTER  := -3;
   const num CMD_TIMEOUT     := -4;
   const num CMD_INVALID_VAL := -5;
   const num CMD_ILL_SYSMODE := -6;
   const num CMD_RES_UNAVAIL := -7;

   ! Predefined modules and files:
   const num HOMEPOS_MODULE  := 10001;
   const num MCPOS_MODULE    := 10002;
   const string SEGMENT_NDX  := "segments.ndx";
   const string NONE_MODULE  := "none";

   ! Filesystem, directories and extensions:
   const string HOME_ROOT       := "HOME:/";
   const string SYSTEM_ROOT     := "INTERNAL:/pntrapid/";
   const string PROGRAM_DIR     := "programs/";
   const string LOG_DIR         := "logs/";
   const string PERS_CONFIG_DIR := "robdata/";
   const string CUST_MAIN_DIR   := "custmain/";
   const string CUST_PNT_DIR    := "custpnt/";
   const string CUST_MC_DIR     := "custmc/";
   const string MODULE_EXT      := ".mod";
   const string SYSMODULE_EXT   := ".sys";

   ! Misc:
   const num IGNORE_MC           := 0;
   const num UNDEFINED_IO_SIG    := -1000000;
   const string SYSTEM_PROC_NAME := "main";

   ! Limits:
   const num MAX_APPLICATORS := 4;

   ! Legacy (commvar.sys stuff For backward compability):
   const string stMedia         := "HOME:";
   const string ST_EMPTY_STRING := "";
   const string ST_PRG_EXT      := ".mod";
   const dionum tpLow           := 0;
   const dionum tpHigh          := 1;
   const dionum tpEdge          := 2;
   const num SYS_UNITIALIZED    := 0;
   const num SYS_DISABLED       := 1;
   const num SYS_STOPPED        := 2;
   const num SYS_READY          := 3;
   const num SYS_IN_PROG_STOP   := 4;
   const num SYS_IN_PROG_RUN    := 5;



endmodule

--- Backups/Robo_open_v2/RAPID/TASK1/SYSMOD/custmain.sys ---
module custmain(sysmodule)



   proc InitCustMain()
      !
      ! This will be executed during startmain/cancel...
      !
      Subscribe PRE_MAIN, "PreMainCustom";
      Subscribe POST_MAIN, "PostMainCustom";
   endproc



   proc PreMainCustom()
      !
      ! This will be executed before a paint program...
      !
   endproc



   proc PostMainCustom()
      !
      ! This will be executed after a paint program...
      !
   endproc



endmodule

--- Backups/Robo_open_v2/RAPID/TASK1/SYSMOD/cycinfo.sys ---
module cycinfo(sysmodule)



   record recCycReport
      string stTag;
      string stInfo;
      string stStart;
      num nDuration;
   endrecord



   local const num MAX_CR_ENTRIES := 15;

   pers recCycReport CurrCycReport{MAX_CR_ENTRIES};
   pers recCycReport LastCycReport{MAX_CR_ENTRIES};

   pers num nCREntriesUsed := 0;



   proc InitCycInfo()
      CycReportRotate; ! Also rotate on cancel.
   endproc



   proc CycReportRotate()
      if nCREntriesUsed > 0 then
         for i from 1 to nCREntriesUsed do
            LastCycReport{i} := CurrCycReport{i};
         endfor
      endif
      for i from (nCREntriesUsed + 1) to Dim(LastCycReport, 1) do
         LastCycReport{i} := ["", "", "", 0];
      endfor

      nCREntriesUsed := 0;
      for i from 1 to Dim(CurrCycReport, 1) do
         CurrCycReport{i} := ["", "", "", 0];
      endfor
   endproc



   local func string stPadToTwo(num nValue)
     if nValue < 10 then
        return "0" + ValToStr(nValue);
     else
        return ValToStr(nValue);
     endif
   endfunc



   local func string stNumToCFormat(num nSeconds)
      var num nMinutes;
      var num nHours;
      var num nMilli;

      nMilli := nSeconds;
      nSeconds := Trunc(nSeconds);
      nMilli := Trunc((nMilli - nSeconds) * 100);

      nHours := nSeconds div 3600;
      nSeconds := nSeconds - (nHours * 3600);
      nMinutes := nSeconds div 60;
      nSeconds := nSeconds - (nMinutes * 60);

      return "0000-00-00 " + stPadToTwo(nHours) + ":" + stPadToTwo(nMinutes) + ":" + stPadToTwo(nSeconds) + "." + stPadToTwo(nMilli);
   endfunc



   proc CycReportUpdate(string stTag \string stStart \string stInfo \num nDuration)
      var num nEntry := -1;

      if stTag = ""
         return;

      ! Does tag exist already?
      for i from 1 to Dim(CurrCycReport, 1) do
         if CurrCycReport{i}.stTag = stTag then
            nEntry := i;
         endif
      endfor

      if nEntry = -1 then
         ! Allocate new tag.
         Incr nCREntriesUsed;
         if nCREntriesUsed > Dim(CurrCycReport, 1) then
            Decr nCREntriesUsed;
            return;
         endif
         nEntry := nCREntriesUsed;
         CurrCycReport{nEntry}.stTag := stTag;
      endif

      if Present(stStart) then
         if RobOS() then
            CurrCycReport{nEntry}.stStart := stStart;
         else
            Set doUpdateVClock;
            WaitDO doUpdateVClock, 0;
            CurrCycReport{nEntry}.stStart := stNumToCFormat(nVirtualClock);
         endif
      endif
      if Present(stInfo)
         CurrCycReport{nEntry}.stInfo := stInfo;
      if Present(nDuration)
         CurrCycReport{nEntry}.nDuration := nDuration;
   endproc



endmodule

--- Backups/Robo_open_v2/RAPID/TASK1/SYSMOD/global.sys ---
module global(sysmodule)
   !
   ! (C) Copyright 2007 ABB
   !



   pers num nCurrProgIndex;
   pers num nCurrMtrlIndex;
   pers num nCurrJobOption;
   pers num nCurrMtrlOption1;
   pers num nCurrMtrlOption2;
   pers bool bCurrExpedited;
   pers num nCurrJobID;

   pers num nDirectProgIndex;
   pers num nDirectJobOption;
   pers bool bDirectExpedited;
   pers string stDirectModule;

   pers string stCurrModule;
   pers num nLastCycleTime;

   pers num nApplicators;

   pers num nRobotState;
   pers num nApplicatorState;
   pers num nProcessState;

   pers num nMasterID{4}; ! 4 = MASTER_CLIENTS constant from master.sys.

   pers num nPntCmdState;
   pers num nGuiSocketPort;
   pers num nVirtualClock;



endmodule

--- Backups/Robo_open_v2/RAPID/TASK1/SYSMOD/qextra.sys ---
module qextra(sysmodule)



   local const num EXTRA_COLUMNS := 3;

   ! Note: Size of the first dimension of this array
   ! have to correspond to the jobqueue size in qdata.sys.
   pers num nExtraQueue{10, EXTRA_COLUMNS} :=
      [[0,0,0],
       [0,0,0],
       [0,0,0],
       [0,0,0],
       [0,0,0],
       [0,0,0],
       [0,0,0],
       [0,0,0],
       [0,0,0],
       [0,0,0]];

   pers num nExtraBuffer{EXTRA_COLUMNS} :=
      [0,0,0];

   pers num nExtraCurrent{EXTRA_COLUMNS} :=
      [0,0,0];



endmodule

--- Backups/Robo_open_v2/RAPID/TASK1/SYSMOD/robdata.sys ---
module robdata(sysmodule)

   ! Note: This file can be used to add custom tools/speeds/zones.
   ! Uncomment any standard tools here, if they are needed.

   ! Robobel 925:
   pers tooldata tRB925_200 := [true,[[290.1,0,540],[0.866025,0,0.5,0]],[8,[0,0,33],[1,0,0,0],0,0,0]];
   pers tooldata tRB925_250 := [true,[[333.4,0,565],[0.866025,0,0.5,0]],[8,[0,0,33],[1,0,0,0],0,0,0]];

   ! HCEBELL:
   pers tooldata tHCEBELL_0   := [true,[[142.9,0,427.5],[0.866025,0,0.5,0]],[10,[0,-40,250],[1,0,0,0],0,0,0]];
   pers tooldata tHCEBELL_150 := [true,[[272.8,0,502.5],[0.866025,0,0.5,0]],[11,[0,40,250],[1,0,0,0],0,0,0]];
   pers tooldata tHCEBELL_200 := [true,[[316.1,0,527.5],[0.866025,0,0.5,0]],[11,[0,40,250],[1,0,0,0],0,0,0]];
   pers tooldata tHCEBELL_250 := [true,[[359.4,0,552.5],[0.866025,0,0.5,0]],[11,[0,40,250],[1,0,0,0],0,0,0]];
   pers tooldata tHCEBELL_300 := [true,[[402.7,0,577.5],[0.866025,0,0.5,0]],[11,[0,40,250],[1,0,0,0],0,0,0]];

   ! Default generic gun (10x5cm, 60 degree):
   pers tooldata tDefGun_Tip := [true,[[50,0,100],[0.866025,0,0.5,0]],[2,[0,0,50],[1,0,0,0],0,0,0]];
   pers tooldata tDefGun_100 := [true,[[136.6,0,150],[0.866025,0,0.5,0]],[2,[0,0,50],[1,0,0,0],0,0,0]];
   pers tooldata tDefGun_200 := [true,[[223.2,0,200],[0.866025,0,0.5,0]],[2,[0,0,50],[1,0,0,0],0,0,0]];

   ! ABB Ecco Gun:
   !pers tooldata tEccoGun_Tip := [true,[[1.8,0,156.6],[0.965926,0,0.258819,0]],[2,[0,0,120],[1,0,0,0],0,0,0]];
   !pers tooldata tEccoGun_200 := [true,[[101.8,0,329.8],[0.965926,0,0.258819,0]],[2,[0,0,120],[1,0,0,0],0,0,0]];
   !pers tooldata tEccoGun_250 := [true,[[126.8,0,373.1],[0.965926,0,0.258819,0]],[2,[0,0,120],[1,0,0,0],0,0,0]];
   !pers tooldata tEccoGun_300 := [true,[[151.8,0,416.4],[0.965926,0,0.258819,0]],[2,[0,0,120],[1,0,0,0],0,0,0]];

   ! G1Direct (short bracket):
   !pers tooldata tG1Direct_300 := [true,[[571.58,0,450],[0.866025,0,0.5,0]],[6.6,[135.2,0,174.1],[1,0,0,0],0,0,0]];
   !pers tooldata tG1Direct_250 := [true,[[528.28,0,425],[0.866025,0,0.5,0]],[6.6,[135.2,0,174.1],[1,0,0,0],0,0,0]];
   !pers tooldata tG1Direct_200 := [true,[[484.97,0,400],[0.866025,0,0.5,0]],[6.6,[135.2,0,174.1],[1,0,0,0],0,0,0]];

   ! G1_Long Braket:
   !pers tooldata tG1V3_200L := [true,[[487,0,502.3],[0.866025,0,0.5,0]],[8,[140.6,0,170],[1,0,0,0],0,0,0]];
   !pers tooldata tG1V3_250L := [true,[[524,0,528.9],[0.866025,0,0.5,0]],[8,[140.6,0,170],[1,0,0,0],0,0,0]];
   !pers tooldata tG1V3_300L := [true,[[549,0,571.6],[0.866025,0,0.5,0]],[8,[140.6,0,170],[1,0,0,0],0,0,0]];

   ! Cartrige Bell:
   !pers tooldata tCBS_0   := [true,[[121.25,0,415],[0.866025,0,0.5,0]],[5.5,[30,0,225],[1,0,0,0],0,0,0]];
   !pers tooldata tCBS_100 := [true,[[207.85,0,465],[0.866025,0,0.5,0]],[5.5,[30,0,225],[1,0,0,0],0,0,0]];
   !pers tooldata tCBS_200 := [true,[[294.45,0,515],[0.866025,0,0.5,0]],[5.5,[30,0,225],[1,0,0,0],0,0,0]];
   !pers tooldata tCBS_250 := [true,[[337.75,0,540],[0.866025,0,0.5,0]],[5.5,[30,0,225],[1,0,0,0],0,0,0]];
   !pers tooldata tCBS_300 := [true,[[381.05,0,565],[0.866025,0,0.5,0]],[5.5,[30,0,225],[1,0,0,0],0,0,0]];

   ! Robobel 926:
   !pers tooldata tRB926TD_0   := [true,[[116.9,0,470],[0.866025,0,0.5,0]],[5.5,[30,0,225],[1,0,0,0],0,0,0]];
   !pers tooldata tRB926TD_100 := [true,[[203.5,0,520],[0.866025,0,0.5,0]],[5.5,[30,0,225],[1,0,0,0],0,0,0]];
   !pers tooldata tRB926TD_120 := [true,[[220.8,0,530],[0.866025,0,0.5,0]],[5.5,[30,0,225],[1,0,0,0],0,0,0]];
   !pers tooldata tRB926TD_150 := [true,[[246.8,0,545],[0.866025,0,0.5,0]],[5.5,[30,0,225],[1,0,0,0],0,0,0]];
   !pers tooldata tRB926TD_200 := [true,[[290.1,0,570],[0.866025,0,0.5,0]],[5.5,[30,0,225],[1,0,0,0],0,0,0]];
   !pers tooldata tRB926TD_250 := [true,[[333.4,0,595],[0.866025,0,0.5,0]],[5.5,[30,0,225],[1,0,0,0],0,0,0]];
   !pers tooldata tRB926TD_300 := [true,[[376.7,0,620],[0.866025,0,0.5,0]],[5.5,[30,0,225],[1,0,0,0],0,0,0]];

   ! Robobel 625TD:
   !pers tooldata tRB625TD_0   := [true,[[116.9,0,420],[0.866025,0,0.5,0]],[5.1,[30,0,215],[1,0,0,0],0,0,0]];
   !pers tooldata tRB625TD_150 := [true,[[246.8,0,495],[0.866025,0,0.5,0]],[5.1,[30,0,215],[1,0,0,0],0,0,0]];
   !pers tooldata tRB625TD_200 := [true,[[290.1,0,520],[0.866025,0,0.5,0]],[5.1,[30,0,215],[1,0,0,0],0,0,0]];
   !pers tooldata tRB625TD_250 := [true,[[333.4,0,545],[0.866025,0,0.5,0]],[5.1,[30,0,215],[1,0,0,0],0,0,0]];
   !pers tooldata tRB625TD_300 := [true,[[376.7,0,570],[0.866025,0,0.5,0]],[5.1,[30,0,215],[1,0,0,0],0,0,0]];

   ! Robobel 951TD:
   !pers tooldata tRB951TD_0   := [true,[[116.9,0,470],[0.866025,0,0.5,0]],[6.3,[30,0,220],[1,0,0,0],0,0,0]];
   !pers tooldata tRB951TD_100 := [true,[[203.5,0,520],[0.866025,0,0.5,0]],[6.3,[30,0,220],[1,0,0,0],0,0,0]];
   !pers tooldata tRB951TD_120 := [true,[[220.8,0,530],[0.866025,0,0.5,0]],[6.3,[30,0,220],[1,0,0,0],0,0,0]];
   !pers tooldata tRB951TD_150 := [true,[[246.8,0,545],[0.866025,0,0.5,0]],[6.3,[30,0,220],[1,0,0,0],0,0,0]];
   !pers tooldata tRB951TD_200 := [true,[[290.1,0,570],[0.866025,0,0.5,0]],[6.3,[30,0,220],[1,0,0,0],0,0,0]];
   !pers tooldata tRB951TD_250 := [true,[[333.4,0,595],[0.866025,0,0.5,0]],[6.3,[30,0,220],[1,0,0,0],0,0,0]];
   !pers tooldata tRB951TD_300 := [true,[[376.7,0,620],[0.866025,0,0.5,0]],[6.3,[30,0,220],[1,0,0,0],0,0,0]];

   ! Robobel 951CBS /40pai/50pai/70pai:
   !pers tooldata tRB951CBS_0   := [true,[[121.25,0,415],[0.866025,0,0.5,0]],[6.3,[55,0,225],[1,0,0,0],0,0,0]];
   !pers tooldata tRB951CBS_100 := [true,[[207.85,0,465],[0.866025,0,0.5,0]],[6.3,[55,0,225],[1,0,0,0],0,0,0]];
   !pers tooldata tRB951CBS_120 := [true,[[225.17,0,475],[0.866025,0,0.5,0]],[6.3,[55,0,225],[1,0,0,0],0,0,0]];
   !pers tooldata tRB951CBS_150 := [true,[[251.15,0,490],[0.866025,0,0.5,0]],[6.3,[55,0,225],[1,0,0,0],0,0,0]];
   !pers tooldata tRB951CBS_200 := [true,[[294.45,0,515],[0.866025,0,0.5,0]],[6.3,[55,0,225],[1,0,0,0],0,0,0]];
   !pers tooldata tRB951CBS_250 := [true,[[337.75,0,540],[0.866025,0,0.5,0]],[6.3,[55,0,225],[1,0,0,0],0,0,0]];
   !pers tooldata tRB951CBS_300 := [true,[[381.05,0,565],[0.866025,0,0.5,0]],[6.3,[55,0,225],[1,0,0,0],0,0,0]];

   ! Interior Robobel951CBS /30pai:
   !pers tooldata tInteriorCBS_0   := [true,[[99.6,0,402.5],[0.866025,0,0.5,0]],[6.3,[30,0,220],[1,0,0,0],0,0,0]];
   !pers tooldata tInteriorCBS_100 := [true,[[186.2,0,452.5],[0.866025,0,0.5,0]],[6.3,[30,0,220],[1,0,0,0],0,0,0]];
   !pers tooldata tInteriorCBS_120 := [true,[[246.8,0,487.5],[0.866025,0,0.5,0]],[6.3,[30,0,220],[1,0,0,0],0,0,0]];
   !pers tooldata tInteriorCBS_150 := [true,[[272.8,0,502.5],[0.866025,0,0.5,0]],[6.3,[30,0,220],[1,0,0,0],0,0,0]];
   !pers tooldata tInteriorCBS_200 := [true,[[316.1,0,527.5],[0.866025,0,0.5,0]],[6.3,[30,0,220],[1,0,0,0],0,0,0]];
   !pers tooldata tInteriorCBS_250 := [true,[[359.4,0,552.5],[0.866025,0,0.5,0]],[6.3,[30,0,220],[1,0,0,0],0,0,0]];
   !pers tooldata tInteriorCBS_300 := [true,[[402.7,0,577.5],[0.866025,0,0.5,0]],[6.3,[30,0,220],[1,0,0,0],0,0,0]];

   ! Interior Robobel951 /30pai:
   !pers tooldata tInterior951_0   := [true,[[138.6,0,482.5],[0.866025,0,0.5,0]],[6.3,[30,0,220],[1,0,0,0],0,0,0]];
   !pers tooldata tInterior951_100 := [true,[[225.17,0,532.5],[0.866025,0,0.5,0]],[6.3,[30,0,220],[1,0,0,0],0,0,0]];
   !pers tooldata tInterior951_120 := [true,[[242.49,0,542.5],[0.866025,0,0.5,0]],[6.3,[30,0,220],[1,0,0,0],0,0,0]];
   !pers tooldata tInterior951_150 := [true,[[268.47,0,557.5],[0.866025,0,0.5,0]],[6.3,[30,0,220],[1,0,0,0],0,0,0]];
   !pers tooldata tInterior951_200 := [true,[[311.77,0,582.5],[0.866025,0,0.5,0]],[6.3,[30,0,220],[1,0,0,0],0,0,0]];
   !pers tooldata tInterior951_250 := [true,[[355.07,0,607.5],[0.866025,0,0.5,0]],[6.3,[30,0,220],[1,0,0,0],0,0,0]];
   !pers tooldata tInterior951_300 := [true,[[398.37,0,632.5],[0.866025,0,0.5,0]],[6.3,[30,0,220],[1,0,0,0],0,0,0]];

   ! RB-1000CBS /1C0341/500ccTank or RB-1000WSC /1C0356/700cc:
   !pers tooldata tRB1000WSC_0     := [true,[[121.25,0,450],[0.866025,0,0.5,0]],[10,[-52,0,270],[1,0,0,0],0,0,0]];
   !pers tooldata tRB1000WSC_100   := [true,[[207.85,0,500],[0.866025,0,0.5,0]],[10,[-52,0,270],[1,0,0,0],0,0,0]];
   !pers tooldata tRB1000WSC_150   := [true,[[251.15,0,525],[0.866025,0,0.5,0]],[10,[-52,0,270],[1,0,0,0],0,0,0]];
   !pers tooldata tRB1000WSC_200   := [true,[[294.45,0,550],[0.866025,0,0.5,0]],[10,[-52,0,270],[1,0,0,0],0,0,0]];
   !pers tooldata tRB1000WSC_250   := [true,[[337.75,0,575],[0.866025,0,0.5,0]],[10,[-52,0,270],[1,0,0,0],0,0,0]];
   !pers tooldata tRB1000WSC_300   := [true,[[381.05,0,600],[0.866025,0,0.5,0]],[10,[-52,0,270],[1,0,0,0],0,0,0]];
   !pers tooldata tRB1000WSC_teach := [true,[[-259.801,0,230],[0.866025,0,0.5,0]],[10,[-52,0,270],[1,0,0,0],0,0,0]];

